C05411=1051.547,373.065,-118.694,173.770,40.070,157.709
C05412=1051.539,372.818,-118.654,173.765,40.065,157.708
C05413=1051.531,372.572,-118.614,173.759,40.059,157.706
C05414=1051.524,372.325,-118.575,173.753,40.054,157.704
C05415=1051.517,372.078,-118.535,173.748,40.048,157.703
C05416=1051.509,371.831,-118.495,173.742,40.043,157.701
C05417=1051.502,371.585,-118.455,173.737,40.037,157.700
C05418=1051.493,371.338,-118.416,173.731,40.032,157.698
C05419=1051.486,371.091,-118.376,173.726,40.027,157.697
C05420=1051.478,370.845,-118.336,173.720,40.021,157.695
C05421=1051.470,370.598,-118.298,173.714,40.015,157.694
C05422=1051.463,370.351,-118.258,173.709,40.010,157.692
C05423=1051.454,370.105,-118.219,173.703,40.005,157.691
C05424=1051.447,369.858,-118.180,173.698,40.000,157.689
C05425=1051.440,369.611,-118.140,173.692,39.994,157.688
C05426=1051.432,369.365,-118.101,173.687,39.989,157.686
C05427=1051.424,369.117,-118.062,173.681,39.984,157.685
C05428=1051.417,368.870,-118.022,173.676,39.978,157.683
C05429=1051.409,368.624,-117.984,173.670,39.974,157.682
C05430=1051.401,368.377,-117.944,173.665,39.968,157.680
C05431=1051.394,368.131,-117.905,173.659,39.963,157.679
C05432=1051.386,367.884,-117.865,173.654,39.958,157.677
C05433=1051.379,367.637,-117.827,173.648,39.952,157.676
C05434=1051.371,367.390,-117.787,173.643,39.947,157.674
C05435=1051.364,367.143,-117.748,173.637,39.942,157.673
C05436=1051.356,366.897,-117.709,173.632,39.937,157.672
C05437=1051.349,366.650,-117.670,173.626,39.931,157.670
C05438=1051.341,366.403,-117.632,173.621,39.926,157.669
C05439=1051.333,366.157,-117.592,173.615,39.921,157.667
C05440=1051.325,365.909,-117.554,173.610,39.916,157.666
C05441=1051.319,365.663,-117.515,173.604,39.911,157.664
C05442=1051.311,365.415,-117.475,173.599,39.906,157.663
C05443=1051.303,365.169,-117.437,173.594,39.900,157.661
C05444=1051.296,364.922,-117.398,173.589,39.895,157.660
C05445=1051.288,364.675,-117.359,173.584,39.890,157.659
C05446=1051.281,364.428,-117.320,173.578,39.885,157.657
C05447=1051.274,364.182,-117.282,173.573,39.880,157.656
C05448=1051.267,363.934,-117.243,173.567,39.875,157.654
C05449=1051.259,363.688,-117.205,173.562,39.870,157.653
C05450=1051.252,363.441,-117.166,173.557,39.865,157.651
C05451=1051.244,363.194,-117.127,173.552,39.860,157.650
C05452=1051.237,362.947,-117.088,173.547,39.855,157.649
C05453=1051.229,362.700,-117.050,173.541,39.850,157.647
C05454=1051.221,362.453,-117.011,173.536,39.845,157.646
C05455=1051.215,362.206,-116.973,173.530,39.840,157.644
C05456=1051.207,361.960,-116.934,173.526,39.835,157.643
C05457=1051.199,361.713,-116.896,173.521,39.830,157.642
C05458=1051.192,361.466,-116.857,173.515,39.825,157.640
C05459=1051.184,361.173,-116.812,173.509,39.819,157.639
C05460=1051.174,360.880,-116.766,173.503,39.813,157.637
C05461=1051.165,360.587,-116.721,173.496,39.808,157.636
C05462=1051.156,360.295,-116.676,173.491,39.802,157.634
C05463=1051.149,360.048,-116.638,173.485,39.797,157.633
C05464=1051.142,359.801,-116.599,173.480,39.792,157.631
C05465=1051.134,359.554,-116.561,173.476,39.787,157.630
C05466=1051.127,359.307,-116.523,173.470,39.782,157.629
C05467=1051.119,359.060,-116.485,173.465,39.777,157.627
C05468=1051.112,358.813,-116.447,173.460,39.773,157.626
C05469=1051.105,358.566,-116.409,173.455,39.768,157.625
C05470=1051.098,358.320,-116.370,173.450,39.763,157.623
C05471=1051.090,358.072,-116.333,173.445,39.758,157.622
C05472=1051.083,357.825,-116.295,173.440,39.753,157.621
C05473=1051.075,357.578,-116.257,173.435,39.748,157.619
C05474=1051.069,357.331,-116.219,173.430,39.744,157.618
C05475=1051.061,357.084,-116.180,173.424,39.739,157.617
C05476=1051.054,356.837,-116.143,173.420,39.734,157.615
C05477=1051.047,356.590,-116.105,173.415,39.729,157.614
C05478=1051.039,356.344,-116.067,173.410,39.725,157.613
C05479=1051.032,356.096,-116.030,173.405,39.720,157.612
C05480=1051.024,355.849,-115.992,173.400,39.715,157.610
C05481=1051.017,355.601,-115.954,173.395,39.710,157.609
C05482=1051.009,355.355,-115.916,173.391,39.706,157.608
C05483=1051.002,355.108,-115.878,173.385,39.701,157.606
C05484=1050.995,354.861,-115.841,173.380,39.696,157.605
C05485=1050.988,354.614,-115.803,173.376,39.692,157.604
C05486=1050.980,354.366,-115.766,173.370,39.687,157.603
C05487=1050.973,354.119,-115.728,173.365,39.682,157.601
C05488=1050.965,353.873,-115.690,173.361,39.678,157.600
C05489=1050.958,353.626,-115.652,173.356,39.673,157.599
C05490=1050.951,353.378,-115.615,173.350,39.668,157.597
C05491=1050.944,353.131,-115.577,173.346,39.664,157.596
C05492=1050.937,352.884,-115.540,173.341,39.659,157.595
C05493=1050.930,352.638,-115.503,173.337,39.655,157.594
C05494=1050.923,352.391,-115.465,173.331,39.650,157.592
C05495=1050.915,352.143,-115.428,173.326,39.646,157.591
C05496=1050.908,351.896,-115.390,173.322,39.641,157.590
C05497=1050.900,351.649,-115.354,173.317,39.637,157.589
C05498=1050.893,351.402,-115.316,173.312,39.632,157.587
C05499=1050.886,351.155,-115.279,173.307,39.627,157.586
C05500=1050.879,350.908,-115.241,173.303,39.622,157.585
C05501=1050.872,350.661,-115.204,173.298,39.618,157.584
C05502=1050.865,350.414,-115.167,173.293,39.614,157.583
C05503=1050.858,350.166,-115.130,173.288,39.609,157.581
C05504=1050.850,349.919,-115.093,173.283,39.605,157.580
C05505=1050.843,349.672,-115.055,173.279,39.600,157.579
C05506=1050.836,349.424,-115.019,173.274,39.596,157.578
C05507=1050.828,349.177,-114.981,173.270,39.591,157.576
C05508=1050.821,348.931,-114.945,173.264,39.587,157.575
C05509=1050.814,348.683,-114.908,173.260,39.582,157.574
C05510=1050.807,348.436,-114.870,173.255,39.578,157.573
C05511=1050.799,348.189,-114.834,173.251,39.574,157.572
C05512=1050.792,347.942,-114.796,173.246,39.569,157.570
C05513=1050.786,347.695,-114.760,173.242,39.565,157.569
C05514=1050.778,347.448,-114.722,173.236,39.560,157.568
C05515=1050.770,347.160,-114.680,173.231,39.555,157.567
C05516=1050.761,346.873,-114.637,173.226,39.550,157.565
C05517=1050.753,346.585,-114.594,173.220,39.545,157.564
C05518=1050.745,346.298,-114.552,173.215,39.540,157.563
C05519=1050.738,346.051,-114.514,173.210,39.535,157.561
C05520=1050.731,345.804,-114.478,173.206,39.531,157.560
C05521=1050.724,345.556,-114.441,173.202,39.527,157.559
C05522=1050.716,345.309,-114.405,173.196,39.522,157.558
C05523=1050.709,345.062,-114.368,173.192,39.518,157.557
C05524=1050.703,344.814,-114.331,173.187,39.514,157.556
C05525=1050.695,344.567,-114.295,173.183,39.509,157.554
C05526=1050.688,344.321,-114.258,173.178,39.506,157.553
C05527=1050.681,344.073,-114.221,173.174,39.501,157.552
C05528=1050.674,343.825,-114.185,173.169,39.497,157.551
C05529=1050.667,343.578,-114.148,173.165,39.493,157.550
C05530=1050.660,343.331,-114.112,173.161,39.488,157.549
C05531=1050.653,343.084,-114.075,173.155,39.484,157.548
C05532=1050.645,342.837,-114.039,173.151,39.479,157.546
C05533=1050.639,342.590,-114.002,173.146,39.475,157.545
C05534=1050.631,342.343,-113.966,173.142,39.471,157.544
C05535=1050.624,342.095,-113.929,173.138,39.467,157.543
C05536=1050.617,341.848,-113.893,173.133,39.463,157.542
C05537=1050.610,341.601,-113.857,173.129,39.458,157.541
C05538=1050.603,341.354,-113.821,173.124,39.455,157.540
C05539=1050.596,341.106,-113.785,173.120,39.450,157.539
C05540=1050.589,340.859,-113.748,173.116,39.446,157.537
C05541=1050.582,340.611,-113.713,173.111,39.442,157.536
C05542=1050.575,340.364,-113.677,173.106,39.438,157.535
C05543=1050.568,340.116,-113.640,173.102,39.433,157.534
C05544=1050.561,339.870,-113.604,173.097,39.430,157.533
C05545=1050.553,339.622,-113.568,173.093,39.425,157.532
C05546=1050.547,339.375,-113.531,173.089,39.421,157.531
C05547=1050.539,339.127,-113.496,173.084,39.417,157.530
C05548=1050.532,338.880,-113.460,173.080,39.413,157.529
C05549=1050.525,338.633,-113.423,173.076,39.409,157.528
C05550=1050.518,338.386,-113.387,173.071,39.404,157.526
C05551=1050.511,338.138,-113.352,173.067,39.401,157.525
C05552=1050.505,337.891,-113.316,173.063,39.396,157.524
C05553=1050.498,337.644,-113.280,173.058,39.392,157.523
C05554=1050.490,337.396,-113.244,173.054,39.388,157.522
C05555=1050.484,337.149,-113.208,173.050,39.384,157.521
C05556=1050.477,336.902,-113.172,173.046,39.380,157.520
C05557=1050.469,336.654,-113.136,173.041,39.376,157.519
C05558=1050.462,336.407,-113.101,173.037,39.372,157.518
C05559=1050.456,336.160,-113.065,173.033,39.368,157.517
C05560=1050.449,335.912,-113.029,173.028,39.364,157.516
C05561=1050.442,335.665,-112.993,173.024,39.360,157.514
C05562=1050.434,335.417,-112.957,173.020,39.356,157.513
C05563=1050.427,335.170,-112.922,173.016,39.352,157.512
C05564=1050.421,334.923,-112.887,173.011,39.348,157.511
C05565=1050.413,334.675,-112.851,173.007,39.344,157.510
C05566=1050.406,334.428,-112.816,173.003,39.340,157.509
C05567=1050.399,334.181,-112.780,172.999,39.336,157.508
C05568=1050.392,333.933,-112.744,172.994,39.332,157.507
C05569=1050.386,333.685,-112.709,172.990,39.328,157.506
C05570=1050.379,333.439,-112.673,172.986,39.324,157.505
C05571=1050.370,333.147,-112.632,172.980,39.319,157.504
C05572=1050.362,332.856,-112.590,172.975,39.315,157.503
C05573=1050.354,332.564,-112.548,172.971,39.310,157.501
C05574=1050.346,332.273,-112.506,172.966,39.306,157.500
C05575=1050.339,332.025,-112.471,172.962,39.302,157.499
C05576=1050.332,331.778,-112.435,172.957,39.297,157.498
C05577=1050.325,331.531,-112.400,172.953,39.293,157.497
C05578=1050.318,331.283,-112.365,172.949,39.290,157.496
C05579=1050.311,331.036,-112.329,172.945,39.286,157.495
C05580=1050.304,330.788,-112.294,172.941,39.282,157.494
C05581=1050.297,330.541,-112.259,172.936,39.278,157.493
C05582=1050.290,330.294,-112.224,172.932,39.274,157.492
C05583=1050.284,330.046,-112.188,172.928,39.270,157.491
C05584=1050.277,329.799,-112.153,172.924,39.266,157.490
C05585=1050.270,329.552,-112.118,172.920,39.262,157.489
C05586=1050.263,329.303,-112.083,172.916,39.258,157.488
C05587=1050.255,329.056,-112.048,172.911,39.255,157.487
C05588=1050.249,328.809,-112.013,172.907,39.251,157.486
C05589=1050.242,328.561,-111.979,172.903,39.247,157.485
C05590=1050.235,328.314,-111.944,172.900,39.244,157.484
C05591=1050.228,328.067,-111.909,172.896,39.240,157.483
C05592=1050.220,327.819,-111.874,172.892,39.236,157.482
C05593=1050.213,327.572,-111.839,172.887,39.232,157.481
C05594=1050.206,327.324,-111.804,172.883,39.229,157.480
C05595=1050.199,327.077,-111.770,172.879,39.225,157.479
C05596=1050.192,326.829,-111.735,172.875,39.221,157.478
C05597=1050.185,326.582,-111.700,172.871,39.217,157.477
C05598=1050.178,326.334,-111.666,172.867,39.213,157.476
C05599=1050.171,326.087,-111.631,172.863,39.210,157.475
C05600=1050.165,325.839,-111.595,172.859,39.206,157.474
C05601=1050.157,325.592,-111.562,172.854,39.202,157.473
C05602=1050.150,325.344,-111.526,172.850,39.199,157.472
C05603=1050.143,325.097,-111.492,172.847,39.195,157.471
C05604=1050.136,324.849,-111.457,172.843,39.191,157.470
C05605=1050.129,324.601,-111.422,172.839,39.188,157.469
C05606=1050.122,324.354,-111.388,172.835,39.184,157.468
C05607=1050.115,324.106,-111.353,172.831,39.180,157.467
C05608=1050.108,323.859,-111.319,172.827,39.177,157.467
C05609=1050.101,323.611,-111.284,172.823,39.173,157.466
C05610=1050.095,323.364,-111.249,172.819,39.169,157.465
C05611=1050.088,323.117,-111.216,172.815,39.166,157.464
C05612=1050.081,322.869,-111.180,172.811,39.162,157.463
C05613=1050.074,322.622,-111.147,172.808,39.158,157.462
C05614=1050.068,322.374,-111.112,172.804,39.154,157.461
C05615=1050.061,322.126,-111.077,172.800,39.151,157.460
C05616=1050.054,321.879,-111.043,172.795,39.147,157.459
C05617=1050.047,321.631,-111.008,172.791,39.144,157.458
C05618=1050.040,321.384,-110.974,172.787,39.140,157.457
C05619=1050.033,321.136,-110.940,172.783,39.136,157.456
C05620=1050.026,320.889,-110.905,172.779,39.132,157.455
C05621=1050.020,320.641,-110.871,172.775,39.129,157.454
C05622=1050.013,320.394,-110.837,172.772,39.125,157.453
C05623=1050.006,320.146,-110.802,172.768,39.121,157.452
C05624=1049.999,319.898,-110.768,172.764,39.118,157.451
C05625=1049.992,319.651,-110.734,172.760,39.114,157.450
C05626=1049.986,319.403,-110.700,172.756,39.110,157.449
C05627=1049.978,319.107,-110.659,172.752,39.106,157.448
C05628=1049.970,318.811,-110.618,172.747,39.102,157.447
C05629=1049.962,318.514,-110.576,172.743,39.098,157.446
C05630=1049.954,318.217,-110.536,172.738,39.093,157.445
C05631=1049.946,317.970,-110.501,172.734,39.090,157.444
C05632=1049.940,317.723,-110.467,172.730,39.086,157.443
C05633=1049.933,317.475,-110.434,172.727,39.083,157.442
C05634=1049.927,317.227,-110.399,172.723,39.079,157.441
C05635=1049.920,316.979,-110.365,172.720,39.075,157.440
C05636=1049.914,316.732,-110.331,172.716,39.072,157.439
C05637=1049.906,316.485,-110.297,172.712,39.068,157.439
C05638=1049.900,316.237,-110.263,172.708,39.064,157.438
C05639=1049.893,315.990,-110.230,172.704,39.061,157.437
C05640=1049.887,315.742,-110.195,172.700,39.057,157.436
C05641=1049.880,315.494,-110.161,172.697,39.054,157.435
C05642=1049.874,315.247,-110.127,172.693,39.050,157.434
C05643=1049.867,314.999,-110.093,172.689,39.047,157.433
C05644=1049.861,314.752,-110.059,172.685,39.043,157.432
C05645=1049.854,314.504,-110.026,172.681,39.039,157.431
C05646=1049.847,314.256,-109.991,172.678,39.035,157.430
C05647=1049.841,314.009,-109.958,172.675,39.032,157.429
C05648=1049.834,313.761,-109.923,172.671,39.029,157.429
C05649=1049.827,313.514,-109.890,172.667,39.025,157.428
C05650=1049.821,313.266,-109.855,172.663,39.022,157.427
C05651=1049.815,313.019,-109.823,172.659,39.018,157.426
C05652=1049.808,312.771,-109.789,172.655,39.014,157.425
C05653=1049.800,312.523,-109.755,172.652,39.011,157.424
C05654=1049.794,312.276,-109.722,172.648,39.008,157.423
C05655=1049.787,312.028,-109.688,172.645,39.004,157.422
C05656=1049.780,311.780,-109.655,172.641,39.001,157.421
C05657=1049.773,311.533,-109.622,172.637,38.997,157.420
C05658=1049.766,311.285,-109.588,172.634,38.994,157.420
C05659=1049.759,311.037,-109.555,172.630,38.991,157.419
C05660=1049.753,310.790,-109.521,172.626,38.987,157.418
C05661=1049.745,310.542,-109.488,172.622,38.984,157.417
C05662=1049.739,310.294,-109.455,172.618,38.981,157.416
C05663=1049.732,310.047,-109.421,172.616,38.977,157.415
C05664=1049.726,309.799,-109.388,172.612,38.974,157.415
C05665=1049.718,309.552,-109.355,172.608,38.971,157.414
C05666=1049.711,309.303,-109.322,172.604,38.967,157.413
C05667=1049.704,309.057,-109.289,172.601,38.964,157.412
C05668=1049.697,308.808,-109.255,172.597,38.961,157.411
C05669=1049.691,308.561,-109.222,172.593,38.957,157.410
C05670=1049.684,308.313,-109.189,172.590,38.953,157.409
C05671=1049.678,308.065,-109.156,172.586,38.950,157.408
C05672=1049.670,307.818,-109.122,172.583,38.947,157.408
C05673=1049.664,307.570,-109.090,172.579,38.943,157.407
C05674=1049.656,307.322,-109.057,172.575,38.940,157.406
C05675=1049.650,307.075,-109.024,172.571,38.937,157.405
C05676=1049.644,306.828,-108.991,172.569,38.933,157.404
C05677=1049.637,306.579,-108.958,172.565,38.930,157.403
C05678=1049.630,306.332,-108.924,172.561,38.927,157.403
C05679=1049.623,306.084,-108.891,172.557,38.923,157.402
C05680=1049.617,305.836,-108.858,172.553,38.920,157.401
C05681=1049.610,305.589,-108.825,172.551,38.917,157.400
C05682=1049.603,305.341,-108.792,172.547,38.913,157.399
C05683=1049.595,305.049,-108.753,172.543,38.909,157.398
C05684=1049.587,304.757,-108.714,172.538,38.905,157.397
C05685=1049.580,304.466,-108.676,172.534,38.901,157.396
C05686=1049.571,304.174,-108.637,172.530,38.898,157.395
C05687=1049.564,303.925,-108.604,172.527,38.894,157.394
C05688=1049.558,303.678,-108.571,172.523,38.891,157.394
C05689=1049.552,303.430,-108.538,172.520,38.887,157.393
C05690=1049.545,303.182,-108.505,172.516,38.884,157.392
C05691=1049.539,302.934,-108.473,172.513,38.881,157.391
C05692=1049.532,302.687,-108.440,172.509,38.877,157.390
C05693=1049.525,302.439,-108.407,172.506,38.875,157.389
C05694=1049.518,302.191,-108.375,172.502,38.871,157.389
C05695=1049.512,301.943,-108.342,172.499,38.868,157.388
C05696=1049.506,301.696,-108.309,172.495,38.865,157.387
C05697=1049.499,301.448,-108.276,172.492,38.861,157.386
C05698=1049.493,301.200,-108.243,172.488,38.858,157.385
C05699=1049.486,300.953,-108.211,172.485,38.854,157.384
C05700=1049.479,300.705,-108.178,172.482,38.851,157.384
C05701=1049.472,300.457,-108.145,172.478,38.848,157.383
C05702=1049.466,300.209,-108.113,172.474,38.844,157.382
C05703=1049.460,299.962,-108.080,172.472,38.841,157.381
C05704=1049.453,299.714,-108.048,172.468,38.838,157.380
C05705=1049.446,299.467,-108.015,172.464,38.835,157.380
C05706=1049.440,299.218,-107.982,172.461,38.831,157.379
C05707=1049.433,298.971,-107.949,172.458,38.828,157.378
C05708=1049.427,298.723,-107.916,172.454,38.825,157.377
C05709=1049.420,298.475,-107.885,172.451,38.821,157.376
C05710=1049.414,298.228,-107.852,172.447,38.818,157.375
C05711=1049.408,297.980,-107.819,172.444,38.815,157.375
C05712=1049.401,297.733,-107.787,172.441,38.812,157.374
C05713=1049.394,297.484,-107.754,172.437,38.808,157.373
C05714=1049.388,297.236,-107.722,172.433,38.805,157.372
C05715=1049.381,296.989,-107.689,172.431,38.802,157.371
C05716=1049.375,296.741,-107.657,172.427,38.798,157.370
C05717=1049.369,296.493,-107.625,172.424,38.795,157.370
C05718=1049.362,296.246,-107.592,172.421,38.792,157.369
C05719=1049.356,295.998,-107.560,172.417,38.789,157.368
C05720=1049.350,295.750,-107.528,172.414,38.785,157.367
C05721=1049.342,295.502,-107.495,172.410,38.782,157.366
C05722=1049.336,295.254,-107.462,172.407,38.779,157.366
C05723=1049.329,295.006,-107.431,172.404,38.776,157.365
C05724=1049.323,294.759,-107.398,172.400,38.772,157.364
C05725=1049.316,294.511,-107.367,172.398,38.770,157.363
C05726=1049.309,294.264,-107.335,172.394,38.766,157.363
C05727=1049.303,294.015,-107.303,172.390,38.763,157.362
C05728=1049.296,293.768,-107.270,172.388,38.760,157.361
C05729=1049.290,293.520,-107.238,172.384,38.757,157.360
C05730=1049.283,293.271,-107.207,172.381,38.753,157.359
C05731=1049.276,293.024,-107.174,172.377,38.750,157.359
C05732=1049.270,292.776,-107.142,172.374,38.747,157.358
C05733=1049.263,292.529,-107.110,172.371,38.744,157.357
C05734=1049.256,292.281,-107.079,172.367,38.741,157.356
C05735=1049.250,292.032,-107.047,172.365,38.737,157.355
C05736=1049.243,291.785,-107.015,172.361,38.735,157.355
C05737=1049.237,291.537,-106.983,172.357,38.731,157.354
C05738=1049.230,291.289,-106.951,172.355,38.729,157.353
C05739=1049.223,291.013,-106.915,172.351,38.725,157.352
C05740=1049.216,290.737,-106.880,172.347,38.721,157.351
C05741=1049.208,290.462,-106.845,172.343,38.718,157.351
C05742=1049.201,290.186,-106.810,172.340,38.714,157.350
C05743=1049.194,289.938,-106.778,172.337,38.711,157.349
C05744=1049.188,289.689,-106.746,172.333,38.708,157.348
C05745=1049.181,289.442,-106.714,172.330,38.705,157.347
C05746=1049.174,289.194,-106.682,172.327,38.702,157.347
C05747=1049.168,288.946,-106.651,172.324,38.699,157.346
C05748=1049.162,288.698,-106.619,172.320,38.696,157.345
C05749=1049.155,288.450,-106.588,172.318,38.692,157.344
C05750=1049.148,288.202,-106.556,172.314,38.690,157.344
C05751=1049.141,287.955,-106.524,172.311,38.686,157.343
C05752=1049.135,287.707,-106.492,172.308,38.683,157.342
C05753=1049.129,287.459,-106.461,172.305,38.680,157.341
C05754=1049.122,287.211,-106.429,172.301,38.677,157.341
C05755=1049.115,286.963,-106.398,172.299,38.674,157.340
C05756=1049.108,286.715,-106.366,172.295,38.671,157.339
C05757=1049.102,286.467,-106.335,172.292,38.667,157.338
C05758=1049.095,286.219,-106.303,172.289,38.665,157.338
C05759=1049.085,285.816,-106.253,172.284,38.660,157.336
C05760=1049.074,285.412,-106.201,172.279,38.654,157.335
C05761=1049.063,285.009,-106.150,172.274,38.650,157.334
C05762=1049.052,284.605,-106.100,172.268,38.645,157.333
C05763=1049.045,284.358,-106.068,172.265,38.641,157.332
C05764=1049.039,284.109,-106.036,172.262,38.639,157.331
C05765=1049.033,283.861,-106.005,172.259,38.636,157.331
C05766=1049.026,283.613,-105.974,172.256,38.632,157.330
C05767=1049.020,283.365,-105.943,172.252,38.630,157.329
C05768=1049.013,283.117,-105.911,172.249,38.626,157.328
C05769=1049.007,282.870,-105.880,172.247,38.623,157.327
C05770=1049.000,282.622,-105.849,172.243,38.621,157.327
C05771=1048.994,282.373,-105.818,172.241,38.617,157.326
C05772=1048.987,282.126,-105.787,172.237,38.614,157.325
C05773=1048.980,281.878,-105.755,172.234,38.611,157.324
C05774=1048.974,281.630,-105.724,172.231,38.608,157.324
C05775=1048.968,281.382,-105.694,172.228,38.605,157.323
C05776=1048.961,281.134,-105.662,172.224,38.602,157.322
C05777=1048.954,280.886,-105.631,172.222,38.599,157.322
C05778=1048.948,280.638,-105.600,172.219,38.595,157.321
C05779=1048.942,280.390,-105.569,172.215,38.593,157.320
C05780=1048.935,280.142,-105.537,172.213,38.590,157.319
C05781=1048.928,279.894,-105.507,172.209,38.586,157.319
C05782=1048.922,279.646,-105.475,172.206,38.584,157.318
C05783=1048.916,279.398,-105.445,172.204,38.580,157.317
C05784=1048.909,279.150,-105.414,172.200,38.577,157.316
C05785=1048.902,278.902,-105.383,172.198,38.574,157.316
C05786=1048.895,278.654,-105.352,172.194,38.572,157.315
C05787=1048.889,278.406,-105.322,172.191,38.568,157.314
C05788=1048.883,278.158,-105.290,172.189,38.565,157.313
C05789=1048.876,277.910,-105.259,172.185,38.563,157.313
C05790=1048.869,277.662,-105.229,172.182,38.560,157.312
C05791=1048.860,277.305,-105.185,172.177,38.555,157.311
C05792=1048.851,276.949,-105.141,172.174,38.551,157.310
C05793=1048.842,276.592,-105.096,172.170,38.547,157.309
C05794=1048.832,276.235,-105.052,172.165,38.542,157.308
C05795=1048.825,275.987,-105.021,172.162,38.539,157.307
C05796=1048.819,275.739,-104.990,172.159,38.536,157.306
C05797=1048.813,275.491,-104.960,172.156,38.533,157.306
C05798=1048.806,275.243,-104.928,172.153,38.530,157.305
C05799=1048.799,274.995,-104.899,172.150,38.527,157.304
C05800=1048.793,274.747,-104.868,172.147,38.524,157.304
C05801=1048.786,274.499,-104.836,172.144,38.521,157.303
C05802=1048.780,274.251,-104.807,172.141,38.518,157.302
C05803=1048.773,274.003,-104.776,172.138,38.515,157.301
C05804=1048.767,273.754,-104.745,172.136,38.512,157.301
C05805=1048.760,273.507,-104.715,172.132,38.509,157.300
C05806=1048.753,273.259,-104.684,172.129,38.506,157.299
C05807=1048.747,273.010,-104.653,172.127,38.503,157.299
C05808=1048.741,272.763,-104.624,172.123,38.500,157.298
C05809=1048.734,272.514,-104.593,172.120,38.497,157.297
C05810=1048.728,272.267,-104.563,172.118,38.494,157.296
C05811=1048.721,272.019,-104.532,172.114,38.491,157.296
C05812=1048.714,271.770,-104.501,172.112,38.488,157.295
C05813=1048.708,271.523,-104.471,172.109,38.485,157.294
C05814=1048.701,271.274,-104.440,172.106,38.483,157.294
C05815=1048.695,271.026,-104.410,172.103,38.480,157.293
C05816=1048.688,270.778,-104.380,172.100,38.476,157.292
C05817=1048.682,270.530,-104.349,172.098,38.473,157.291
C05818=1048.675,270.282,-104.320,172.094,38.471,157.291
C05819=1048.669,270.034,-104.289,172.091,38.468,157.290
C05820=1048.662,269.786,-104.259,172.089,38.465,157.289
C05821=1048.656,269.538,-104.228,172.085,38.462,157.289
C05822=1048.649,269.290,-104.198,172.082,38.459,157.288
C05823=1048.643,269.042,-104.168,172.080,38.456,157.287
C05824=1048.636,268.794,-104.138,172.077,38.453,157.287
C05825=1048.630,268.546,-104.107,172.074,38.450,157.286
C05826=1048.623,268.297,-104.077,172.071,38.447,157.285
C05827=1048.617,268.050,-104.047,172.069,38.444,157.284
C05828=1048.610,267.801,-104.018,172.066,38.441,157.284
C05829=1048.604,267.553,-103.988,172.062,38.438,157.283
C05830=1048.597,267.305,-103.957,172.060,38.435,157.282
C05831=1048.591,267.057,-103.927,172.057,38.432,157.282
C05832=1048.584,266.809,-103.897,172.055,38.429,157.281
C05833=1048.578,266.561,-103.868,172.051,38.426,157.280
C05834=1048.571,266.312,-103.837,172.048,38.424,157.280
C05835=1048.564,266.065,-103.808,172.046,38.421,157.279
C05836=1048.558,265.816,-103.777,172.043,38.418,157.278
C05837=1048.551,265.569,-103.747,172.040,38.415,157.278
C05838=1048.545,265.320,-103.717,172.037,38.412,157.277
C05839=1048.539,265.072,-103.687,172.034,38.409,157.276
C05840=1048.532,264.824,-103.657,172.032,38.406,157.275
C05841=1048.526,264.576,-103.628,172.029,38.403,157.275
C05842=1048.519,264.327,-103.598,172.026,38.400,157.274
C05843=1048.512,264.080,-103.568,172.023,38.397,157.273
C05844=1048.506,263.831,-103.538,172.020,38.394,157.273
C05845=1048.500,263.583,-103.508,172.018,38.391,157.272
C05846=1048.493,263.336,-103.478,172.015,38.388,157.271
C05847=1048.486,263.075,-103.447,172.012,38.385,157.271
C05848=1048.480,262.814,-103.416,172.009,38.382,157.270
C05849=1048.473,262.555,-103.385,172.006,38.379,157.269
C05850=1048.466,262.294,-103.354,172.003,38.376,157.268
C05851=1048.459,262.046,-103.324,172.000,38.374,157.268
C05852=1048.453,261.798,-103.295,171.998,38.371,157.267
C05853=1048.446,261.550,-103.264,171.995,38.368,157.266
C05854=1048.439,261.302,-103.235,171.992,38.365,157.266
C05855=1048.433,261.054,-103.206,171.989,38.362,157.265
C05856=1048.426,260.805,-103.176,171.986,38.359,157.264
C05857=1048.419,260.558,-103.146,171.984,38.356,157.264
C05858=1048.413,260.309,-103.117,171.981,38.353,157.263
C05859=1048.406,260.061,-103.088,171.979,38.351,157.262
C05860=1048.399,259.813,-103.058,171.975,38.348,157.262
C05861=1048.393,259.564,-103.029,171.973,38.345,157.261
C05862=1048.386,259.317,-103.000,171.970,38.342,157.260
C05863=1048.379,259.068,-102.970,171.967,38.339,157.260
C05864=1048.373,258.820,-102.941,171.965,38.336,157.259
C05865=1048.366,258.571,-102.912,171.962,38.333,157.258
C05866=1048.359,258.324,-102.882,171.959,38.330,157.258
C05867=1048.353,258.076,-102.853,171.956,38.327,157.257
C05868=1048.346,257.827,-102.824,171.954,38.325,157.256
C05869=1048.339,257.580,-102.794,171.951,38.322,157.256
C05870=1048.333,257.331,-102.765,171.949,38.319,157.255
C05871=1048.326,257.083,-102.735,171.946,38.317,157.254
C05872=1048.320,256.834,-102.706,171.943,38.314,157.254
C05873=1048.314,256.587,-102.677,171.940,38.311,157.253
C05874=1048.307,256.338,-102.647,171.937,38.308,157.252
C05875=1048.300,256.090,-102.618,171.935,38.305,157.252
C05876=1048.294,255.842,-102.589,171.932,38.302,157.251
C05877=1048.287,255.593,-102.560,171.930,38.299,157.250
C05878=1048.281,255.345,-102.530,171.927,38.296,157.250
C05879=1048.275,255.097,-102.501,171.925,38.293,157.249
C05880=1048.268,254.850,-102.472,171.922,38.290,157.248
C05881=1048.261,254.601,-102.443,171.919,38.288,157.248
C05882=1048.254,254.353,-102.414,171.916,38.285,157.247
C05883=1048.248,254.104,-102.385,171.913,38.282,157.246
C05884=1048.242,253.856,-102.356,171.911,38.279,157.246
C05885=1048.235,253.607,-102.327,171.908,38.276,157.245
C05886=1048.229,253.359,-102.298,171.906,38.273,157.244
C05887=1048.222,253.112,-102.268,171.903,38.270,157.244
C05888=1048.216,252.864,-102.239,171.900,38.267,157.243
C05889=1048.209,252.615,-102.209,171.898,38.264,157.242
C05890=1048.203,252.367,-102.180,171.895,38.262,157.242
C05891=1048.196,252.119,-102.152,171.893,38.259,157.241
C05892=1048.190,251.871,-102.123,171.890,38.256,157.240
C05893=1048.183,251.623,-102.094,171.888,38.253,157.240
C05894=1048.177,251.374,-102.064,171.885,38.250,157.239
C05895=1048.170,251.126,-102.035,171.883,38.247,157.238
C05896=1048.164,250.878,-102.006,171.880,38.244,157.238
C05897=1048.158,250.629,-101.977,171.876,38.241,157.237
C05898=1048.152,250.381,-101.949,171.874,38.238,157.236
C05899=1048.146,250.133,-101.920,171.871,38.235,157.236
C05900=1048.138,249.884,-101.891,171.869,38.233,157.235
C05901=1048.132,249.636,-101.862,171.866,38.230,157.234
C05902=1048.126,249.388,-101.833,171.864,38.227,157.234
C05903=1048.119,249.126,-101.802,171.861,38.224,157.233
C05904=1048.113,248.864,-101.772,171.858,38.220,157.232
C05905=1048.106,248.603,-101.741,171.856,38.217,157.231
C05906=1048.098,248.341,-101.711,171.853,38.214,157.231
C05907=1048.092,248.092,-101.683,171.851,38.212,157.230
C05908=1048.086,247.844,-101.653,171.848,38.209,157.229
C05909=1048.080,247.596,-101.624,171.846,38.206,157.229
C05910=1048.074,247.348,-101.595,171.843,38.203,157.228
C05911=1048.067,247.100,-101.566,171.841,38.200,157.227
C05912=1048.062,246.851,-101.538,171.838,38.196,157.227
C05913=1048.055,246.603,-101.510,171.835,38.194,157.226
C05914=1048.048,246.355,-101.481,171.833,38.191,157.225
C05915=1048.042,246.107,-101.451,171.830,38.188,157.225
C05916=1048.036,245.858,-101.423,171.828,38.185,157.224
C05917=1048.030,245.610,-101.394,171.825,38.182,157.223
C05918=1048.022,245.362,-101.365,171.823,38.179,157.223
C05919=1048.016,245.113,-101.337,171.820,38.176,157.222
C05920=1048.010,244.865,-101.308,171.817,38.173,157.221
C05921=1048.003,244.617,-101.280,171.815,38.170,157.221
C05922=1047.997,244.368,-101.251,171.812,38.168,157.220
C05923=1047.990,244.120,-101.223,171.810,38.165,157.219
C05924=1047.984,243.872,-101.194,171.807,38.162,157.219
C05925=1047.978,243.623,-101.165,171.805,38.159,157.218
C05926=1047.971,243.376,-101.137,171.803,38.156,157.217
C05927=1047.965,243.127,-101.109,171.801,38.153,157.217
C05928=1047.958,242.879,-101.080,171.798,38.150,157.216
C05929=1047.952,242.630,-101.052,171.796,38.147,157.215
C05930=1047.946,242.382,-101.023,171.793,38.145,157.215
C05931=1047.939,242.134,-100.995,171.791,38.142,157.214
C05932=1047.933,241.886,-100.966,171.788,38.139,157.213
C05933=1047.926,241.637,-100.938,171.785,38.136,157.213
C05934=1047.920,241.389,-100.909,171.783,38.133,157.212
C05935=1047.913,241.141,-100.882,171.780,38.130,157.211
C05936=1047.907,240.892,-100.853,171.778,38.127,157.211
C05937=1047.900,240.644,-100.825,171.775,38.124,157.210
C05938=1047.894,240.396,-100.797,171.773,38.121,157.209
C05939=1047.887,240.147,-100.768,171.770,38.119,157.209
C05940=1047.881,239.899,-100.740,171.768,38.116,157.208
C05941=1047.874,239.651,-100.713,171.766,38.113,157.208
C05942=1047.868,239.402,-100.683,171.764,38.110,157.207
C05943=1047.861,239.154,-100.656,171.761,38.107,157.206
C05944=1047.855,238.905,-100.627,171.759,38.104,157.206
C05945=1047.848,238.657,-100.599,171.756,38.101,157.205
C05946=1047.842,238.409,-100.571,171.753,38.098,157.204
C05947=1047.836,238.160,-100.543,171.751,38.095,157.204
C05948=1047.829,237.912,-100.515,171.748,38.093,157.203
C05949=1047.822,237.664,-100.487,171.746,38.090,157.202
C05950=1047.815,237.415,-100.459,171.743,38.087,157.202
C05951=1047.809,237.167,-100.431,171.742,38.084,157.201
C05952=1047.803,236.918,-100.403,171.739,38.081,157.200
C05953=1047.796,236.670,-100.375,171.737,38.078,157.200
C05954=1047.790,236.422,-100.346,171.734,38.076,157.199
C05955=1047.783,236.173,-100.318,171.732,38.073,157.198
C05956=1047.777,235.926,-100.291,171.729,38.070,157.198
C05957=1047.770,235.677,-100.263,171.727,38.067,157.197
C05958=1047.764,235.428,-100.235,171.724,38.064,157.197
C05959=1047.757,235.161,-100.205,171.722,38.061,157.196
C05960=1047.749,234.893,-100.175,171.719,38.058,157.195
C05961=1047.743,234.626,-100.145,171.716,38.055,157.195
C05962=1047.736,234.358,-100.115,171.714,38.052,157.194
C05963=1047.730,234.109,-100.087,171.712,38.049,157.193
C05964=1047.723,233.862,-100.059,171.710,38.046,157.192
C05965=1047.717,233.614,-100.031,171.707,38.043,157.192
C05966=1047.711,233.365,-100.003,171.705,38.040,157.191
C05967=1047.704,233.117,-99.975,171.702,38.037,157.191
C05968=1047.697,232.868,-99.947,171.701,38.034,157.190
C05969=1047.691,232.620,-99.920,171.698,38.032,157.189
C05970=1047.685,232.371,-99.891,171.696,38.029,157.189
C05971=1047.679,232.123,-99.864,171.693,38.026,157.188
C05972=1047.672,231.875,-99.836,171.691,38.023,157.187
C05973=1047.665,231.626,-99.808,171.688,38.020,157.187
C05974=1047.658,231.378,-99.781,171.687,38.017,157.186
C05975=1047.652,231.129,-99.753,171.684,38.014,157.185
C05976=1047.645,230.881,-99.725,171.681,38.011,157.185
C05977=1047.640,230.632,-99.698,171.679,38.008,157.184
C05978=1047.633,230.384,-99.670,171.676,38.005,157.183
C05979=1047.627,230.135,-99.642,171.675,38.002,157.183
C05980=1047.620,229.887,-99.615,171.672,38.000,157.182
C05981=1047.613,229.638,-99.587,171.670,37.997,157.181
C05982=1047.607,229.391,-99.560,171.667,37.994,157.181
C05983=1047.601,229.142,-99.532,171.665,37.991,157.180
C05984=1047.594,228.894,-99.504,171.663,37.988,157.180
C05985=1047.588,228.645,-99.477,171.661,37.985,157.179
C05986=1047.581,228.397,-99.450,171.658,37.982,157.178
C05987=1047.575,228.149,-99.422,171.656,37.979,157.178
C05988=1047.568,227.900,-99.394,171.653,37.976,157.177
C05989=1047.562,227.651,-99.367,171.652,37.974,157.176
C05990=1047.555,227.403,-99.340,171.649,37.971,157.176
C05991=1047.549,227.155,-99.312,171.647,37.968,157.175
C05992=1047.542,226.907,-99.285,171.644,37.965,157.174
C05993=1047.535,226.658,-99.258,171.643,37.962,157.174
C05994=1047.528,226.409,-99.230,171.640,37.959,157.173
C05995=1047.522,226.161,-99.203,171.638,37.956,157.172
C05996=1047.516,225.913,-99.176,171.635,37.953,157.172
C05997=1047.509,225.664,-99.148,171.634,37.950,157.171
C05998=1047.503,225.416,-99.121,171.631,37.948,157.171
C05999=1047.497,225.167,-99.094,171.629,37.945,157.170
C06000=1047.490,224.919,-99.066,171.626,37.942,157.169
C06001=1047.484,224.670,-99.039,171.625,37.939,157.169
C06002=1047.476,224.422,-99.012,171.622,37.936,157.168
C06003=1047.470,224.174,-98.985,171.620,37.933,157.167
C06004=1047.464,223.925,-98.958,171.617,37.930,157.167
C06005=1047.457,223.676,-98.930,171.616,37.927,157.166
C06006=1047.452,223.428,-98.903,171.613,37.924,157.165
C06007=1047.445,223.180,-98.875,171.611,37.921,157.165
C06008=1047.438,222.931,-98.848,171.609,37.918,157.164
C06009=1047.432,222.683,-98.822,171.606,37.916,157.163
C06010=1047.425,222.435,-98.794,171.604,37.913,157.163
C06011=1047.419,222.186,-98.767,171.602,37.910,157.162
C06012=1047.412,221.938,-98.740,171.600,37.907,157.162
C06013=1047.406,221.689,-98.713,171.598,37.904,157.161
C06014=1047.399,221.440,-98.685,171.595,37.901,157.160
C06015=1047.392,221.165,-98.655,171.592,37.898,157.159
C06016=1047.385,220.890,-98.625,171.591,37.895,157.159
C06017=1047.378,220.615,-98.595,171.588,37.891,157.158
C06018=1047.371,220.340,-98.566,171.586,37.888,157.157
C06019=1047.365,220.092,-98.539,171.583,37.885,157.157
C06020=1047.358,219.844,-98.511,171.582,37.882,157.156
C06021=1047.351,219.595,-98.485,171.579,37.879,157.155
C06022=1047.345,219.346,-98.458,171.577,37.876,157.155
C06023=1047.338,219.098,-98.431,171.574,37.874,157.154
C06024=1047.331,218.849,-98.404,171.573,37.871,157.153
C06025=1047.326,218.601,-98.377,171.570,37.868,157.153
C06026=1047.318,218.353,-98.350,171.568,37.865,157.152
C06027=1047.312,218.104,-98.323,171.566,37.862,157.152
C06028=1047.305,217.856,-98.297,171.564,37.859,157.151
C06029=1047.299,217.607,-98.270,171.561,37.856,157.150
C06030=1047.293,217.359,-98.243,171.560,37.853,157.150
C06031=1047.286,217.110,-98.216,171.557,37.850,157.149
C06032=1047.279,216.861,-98.189,171.555,37.847,157.148
C06033=1047.273,216.613,-98.163,171.553,37.844,157.148
C06034=1047.266,216.365,-98.135,171.551,37.842,157.147
C06035=1047.260,216.116,-98.109,171.549,37.839,157.146
C06036=1047.253,215.867,-98.082,171.547,37.836,157.146
C06037=1047.248,215.619,-98.056,171.544,37.833,157.145
C06038=1047.240,215.371,-98.029,171.543,37.830,157.145
C06039=1047.234,215.122,-98.002,171.540,37.827,157.144
C06040=1047.227,214.874,-97.976,171.538,37.824,157.143
C06041=1047.221,214.625,-97.949,171.536,37.821,157.143
C06042=1047.214,214.377,-97.922,171.534,37.818,157.142
C06043=1047.208,214.128,-97.895,171.532,37.815,157.141
C06044=1047.202,213.880,-97.868,171.530,37.812,157.141
C06045=1047.195,213.631,-97.842,171.527,37.809,157.140
C06046=1047.189,213.383,-97.815,171.526,37.807,157.139
C06047=1047.182,213.134,-97.789,171.523,37.804,157.139
C06048=1047.176,212.886,-97.762,171.522,37.801,157.138
C06049=1047.169,212.637,-97.736,171.519,37.798,157.137
C06050=1047.163,212.389,-97.709,171.517,37.795,157.137
C06051=1047.156,212.140,-97.682,171.515,37.792,157.136
C06052=1047.150,211.891,-97.656,171.513,37.789,157.136
C06053=1047.143,211.643,-97.629,171.511,37.786,157.135
C06054=1047.137,211.394,-97.603,171.509,37.783,157.134
C06055=1047.130,211.146,-97.576,171.506,37.780,157.134
C06056=1047.124,210.898,-97.550,171.505,37.777,157.133
C06057=1047.117,210.648,-97.523,171.502,37.774,157.132
C06058=1047.111,210.400,-97.497,171.501,37.771,157.132
C06059=1047.105,210.151,-97.470,171.498,37.768,157.131
C06060=1047.098,209.903,-97.444,171.497,37.765,157.130
C06061=1047.092,209.655,-97.418,171.494,37.762,157.130
C06062=1047.085,209.406,-97.391,171.492,37.759,157.129
C06063=1047.079,209.158,-97.365,171.490,37.756,157.128
C06064=1047.072,208.909,-97.339,171.488,37.753,157.128
C06065=1047.066,208.661,-97.312,171.486,37.750,157.127
C06066=1047.059,208.412,-97.286,171.484,37.747,157.126
C06067=1047.052,208.164,-97.260,171.482,37.744,157.126
C06068=1047.046,207.915,-97.233,171.480,37.741,157.125
C06069=1047.040,207.667,-97.207,171.477,37.738,157.125
C06070=1047.033,207.418,-97.181,171.476,37.735,157.124
C06071=1047.026,207.148,-97.153,171.473,37.732,157.123
C06072=1047.019,206.879,-97.124,171.471,37.729,157.122
C06073=1047.011,206.610,-97.096,171.469,37.726,157.122
C06074=1047.004,206.339,-97.067,171.466,37.723,157.121
C06075=1046.978,205.288,-96.961,171.219,37.623,157.097
C06076=1046.972,205.039,-96.936,171.216,37.621,157.097
C06077=1046.966,204.791,-96.911,171.213,37.619,157.097
C06078=1046.960,204.542,-96.886,171.211,37.617,157.096
C06079=1046.954,204.293,-96.861,171.208,37.614,157.095
C06080=1046.948,204.044,-96.836,171.205,37.612,157.095
C06081=1046.942,203.796,-96.810,171.203,37.610,157.095
C06082=1046.936,203.547,-96.785,171.200,37.608,157.094
C06083=1046.930,203.298,-96.761,171.197,37.606,157.094
C06084=1046.924,203.050,-96.735,171.194,37.604,157.093
C06085=1046.918,202.801,-96.710,171.192,37.601,157.093
C06086=1046.911,202.553,-96.685,171.189,37.599,157.092
C06087=1046.906,202.304,-96.661,171.186,37.597,157.092
C06088=1046.900,202.056,-96.636,171.184,37.595,157.091
C06089=1046.893,201.807,-96.610,171.181,37.593,157.091
C06090=1046.887,201.558,-96.586,171.178,37.591,157.090
C06091=1046.881,201.309,-96.560,171.176,37.589,157.090
C06092=1046.876,201.060,-96.536,171.173,37.586,157.089
C06093=1046.869,200.812,-96.511,171.170,37.585,157.089
C06094=1046.863,200.563,-96.487,171.168,37.582,157.088
C06095=1046.856,200.314,-96.462,171.165,37.580,157.088
C06096=1046.850,200.065,-96.438,171.162,37.578,157.088
C06097=1046.845,199.817,-96.413,171.160,37.576,157.087
C06098=1046.838,199.568,-96.389,171.157,37.574,157.087
C06099=1046.832,199.319,-96.363,171.154,37.572,157.086
C06100=1046.825,199.070,-96.339,171.152,37.570,157.086
C06101=1046.819,198.822,-96.314,171.150,37.568,157.085
C06102=1046.814,198.573,-96.290,171.146,37.566,157.085
C06103=1046.807,198.325,-96.265,171.144,37.564,157.084
C06104=1046.801,198.076,-96.240,171.142,37.562,157.084
C06105=1046.794,197.827,-96.215,171.138,37.560,157.084
C06106=1046.789,197.579,-96.191,171.136,37.558,157.083
C06107=1046.782,197.330,-96.167,171.134,37.556,157.083
C06108=1046.776,197.081,-96.142,171.130,37.554,157.082
C06109=1046.770,196.832,-96.118,171.128,37.551,157.082
C06110=1046.764,196.584,-96.093,171.126,37.550,157.081
C06111=1046.758,196.335,-96.068,171.123,37.548,157.081
C06112=1046.752,196.086,-96.045,171.120,37.546,157.080
C06113=1046.745,195.838,-96.019,171.118,37.544,157.080
C06114=1046.739,195.589,-95.995,171.115,37.541,157.080
C06115=1046.733,195.340,-95.971,171.113,37.540,157.079
C06116=1046.727,195.092,-95.946,171.110,37.538,157.079
C06117=1046.721,194.843,-95.922,171.107,37.535,157.078
C06118=1046.715,194.594,-95.897,171.105,37.534,157.078
C06119=1046.709,194.345,-95.873,171.102,37.531,157.077
C06120=1046.702,194.096,-95.848,171.099,37.530,157.077
C06121=1046.696,193.848,-95.824,171.097,37.528,157.077
C06122=1046.691,193.599,-95.800,171.095,37.525,157.076
C06123=1046.684,193.350,-95.776,171.091,37.524,157.076
C06124=1046.678,193.102,-95.751,171.089,37.522,157.075
C06125=1046.672,192.853,-95.727,171.087,37.519,157.075
C06126=1046.666,192.604,-95.702,171.085,37.518,157.074
C06127=1046.660,192.355,-95.678,171.082,37.515,157.074
C06128=1046.654,192.106,-95.654,171.079,37.513,157.074
C06129=1046.648,191.858,-95.629,171.077,37.512,157.073
C06130=1046.642,191.609,-95.605,171.074,37.509,157.073
C06131=1046.636,191.360,-95.580,171.072,37.508,157.072
C06132=1046.630,191.111,-95.556,171.069,37.506,157.072
C06133=1046.624,190.863,-95.532,171.066,37.503,157.071
C06134=1046.618,190.614,-95.508,171.064,37.502,157.071
C06135=1046.612,190.365,-95.484,171.062,37.500,157.071
C06136=1046.605,190.081,-95.456,171.058,37.497,157.070
C06137=1046.598,189.796,-95.428,171.056,37.495,157.070
C06138=1046.591,189.512,-95.400,171.053,37.493,157.069
C06139=1046.584,189.228,-95.373,171.050,37.490,157.069
C06140=1046.578,188.979,-95.349,171.048,37.488,157.068
C06141=1046.572,188.730,-95.325,171.045,37.487,157.068
C06142=1046.566,188.481,-95.300,171.042,37.484,157.067
C06143=1046.560,188.233,-95.277,171.040,37.483,157.067
C06144=1046.554,187.983,-95.252,171.038,37.481,157.066
C06145=1046.548,187.735,-95.229,171.035,37.478,157.066
C06146=1046.542,187.486,-95.204,171.032,37.477,157.066
C06147=1046.536,187.238,-95.180,171.030,37.475,157.065
C06148=1046.531,186.988,-95.156,171.027,37.473,157.065
C06149=1046.524,186.740,-95.132,171.025,37.471,157.064
C06150=1046.519,186.491,-95.108,171.023,37.469,157.064
C06151=1046.513,186.242,-95.084,171.020,37.467,157.063
C06152=1046.507,185.994,-95.059,171.018,37.465,157.063
C06153=1046.501,185.745,-95.035,171.015,37.463,157.063
C06154=1046.495,185.496,-95.011,171.013,37.461,157.062
C06155=1046.489,185.247,-94.987,171.010,37.459,157.062
C06156=1046.484,184.998,-94.964,171.008,37.457,157.061
C06157=1046.478,184.750,-94.940,171.006,37.455,157.061
C06158=1046.472,184.501,-94.915,171.003,37.453,157.061
C06159=1046.466,184.252,-94.892,171.001,37.451,157.060
C06160=1046.460,184.003,-94.867,170.998,37.449,157.060
C06161=1046.454,183.755,-94.843,170.995,37.447,157.059
C06162=1046.448,183.506,-94.820,170.993,37.446,157.059
C06163=1046.441,183.257,-94.796,170.991,37.444,157.059
C06164=1046.435,183.009,-94.773,170.989,37.442,157.058
C06165=1046.429,182.759,-94.749,170.986,37.440,157.058
C06166=1046.423,182.511,-94.726,170.983,37.438,157.057
C06167=1046.416,182.262,-94.702,170.981,37.437,157.057
C06168=1046.410,182.013,-94.679,170.978,37.435,157.057
C06169=1046.403,181.764,-94.655,170.976,37.433,157.056
C06170=1046.397,181.516,-94.632,170.974,37.431,157.056
C06171=1046.391,181.266,-94.608,170.972,37.429,157.055
C06172=1046.385,181.018,-94.585,170.968,37.428,157.055
C06173=1046.379,180.768,-94.561,170.966,37.426,157.055
C06174=1046.372,180.520,-94.538,170.964,37.424,157.054
C06175=1046.366,180.271,-94.514,170.961,37.422,157.054
C06176=1046.360,180.022,-94.491,170.959,37.421,157.054
C06177=1046.354,179.774,-94.467,170.957,37.419,157.053
C06178=1046.348,179.524,-94.444,170.954,37.417,157.053
C06179=1046.342,179.276,-94.420,170.951,37.415,157.052
C06180=1046.335,179.026,-94.397,170.949,37.413,157.052
C06181=1046.329,178.779,-94.374,170.947,37.412,157.052
C06182=1046.323,178.530,-94.351,170.945,37.410,157.051
C06183=1046.316,178.281,-94.327,170.942,37.408,157.051
C06184=1046.311,178.032,-94.304,170.940,37.406,157.050
C06185=1046.304,177.783,-94.280,170.938,37.404,157.050
C06186=1046.298,177.534,-94.257,170.934,37.403,157.050
C06187=1046.292,177.286,-94.233,170.932,37.401,157.049
C06188=1046.286,177.036,-94.210,170.930,37.400,157.049
C06189=1046.280,176.788,-94.186,170.928,37.398,157.049
C06190=1046.274,176.539,-94.163,170.925,37.396,157.048
C06191=1046.267,176.290,-94.141,170.923,37.394,157.048
C06192=1046.261,176.041,-94.117,170.921,37.392,157.048
C06193=1046.255,175.792,-94.094,170.919,37.391,157.047
C06194=1046.249,175.543,-94.070,170.916,37.389,157.047
C06195=1046.243,175.294,-94.047,170.913,37.387,157.046
C06196=1046.237,175.046,-94.024,170.911,37.385,157.046
C06197=1046.231,174.797,-94.000,170.908,37.383,157.046
C06198=1046.225,174.548,-93.977,170.906,37.382,157.045
C06199=1046.219,174.299,-93.954,170.904,37.380,157.045
C06200=1046.213,174.083,-93.934,170.902,37.379,157.045
C06201=1046.209,173.869,-93.914,170.900,37.377,157.044
C06202=1046.202,173.654,-93.894,170.898,37.376,157.044
C06203=1046.197,173.438,-93.874,170.896,37.374,157.044
C06204=1046.192,173.224,-93.854,170.894,37.373,157.043
C06205=1046.187,173.008,-93.834,170.892,37.371,157.043
C06206=1046.181,172.793,-93.814,170.890,37.370,157.043
C06207=1046.176,172.578,-93.794,170.888,37.368,157.042
C06208=1046.171,172.329,-93.771,170.886,37.366,157.042
C06209=1046.164,172.080,-93.748,170.884,37.364,157.042
C06210=1046.158,171.831,-93.724,170.881,37.363,157.041
C06211=1046.152,171.582,-93.701,170.879,37.361,157.041
C06212=1046.147,171.334,-93.678,170.877,37.359,157.040
C06213=1046.140,171.085,-93.656,170.873,37.357,157.040
C06214=1046.134,170.836,-93.632,170.871,37.356,157.040
C06215=1046.128,170.587,-93.609,170.869,37.354,157.039
C06216=1046.122,170.338,-93.586,170.867,37.352,157.039
C06217=1046.116,170.089,-93.563,170.864,37.351,157.039
C06218=1046.111,169.840,-93.540,170.862,37.349,157.038
C06219=1046.104,169.591,-93.516,170.860,37.347,157.038
C06220=1046.098,169.343,-93.494,170.858,37.345,157.037
C06221=1046.092,169.094,-93.471,170.855,37.343,157.037
C06222=1046.086,168.845,-93.448,170.853,37.342,157.037
C06223=1046.080,168.596,-93.425,170.851,37.340,157.036
C06224=1046.075,168.347,-93.402,170.849,37.338,157.036
C06225=1046.069,168.098,-93.379,170.846,37.337,157.036
C06226=1046.062,167.849,-93.356,170.844,37.335,157.035
C06227=1046.056,167.601,-93.333,170.842,37.333,157.035
C06228=1046.050,167.352,-93.310,170.840,37.331,157.035
C06229=1046.044,167.103,-93.287,170.837,37.330,157.034
C06230=1046.039,166.854,-93.264,170.835,37.328,157.034
C06231=1046.032,166.606,-93.241,170.833,37.326,157.033
C06232=1046.026,166.357,-93.218,170.830,37.324,157.033
C06233=1046.021,166.108,-93.195,170.828,37.322,157.033
C06234=1046.015,165.859,-93.172,170.826,37.320,157.032
C06235=1046.009,165.610,-93.150,170.824,37.319,157.032
C06236=1046.002,165.361,-93.127,170.821,37.317,157.032
C06237=1045.996,165.112,-93.104,170.819,37.316,157.031
C06238=1045.991,164.863,-93.081,170.817,37.314,157.031
C06239=1045.985,164.614,-93.058,170.815,37.312,157.030
C06240=1045.977,164.262,-93.026,170.811,37.310,157.030
C06241=1045.968,163.910,-92.994,170.809,37.307,157.029
C06242=1045.960,163.558,-92.961,170.806,37.305,157.029
C06243=1045.952,163.205,-92.929,170.802,37.302,157.028
C06244=1045.946,162.956,-92.906,170.800,37.301,157.028
C06245=1045.940,162.707,-92.884,170.798,37.299,157.028
C06246=1045.934,162.458,-92.861,170.795,37.297,157.027
C06247=1045.928,162.210,-92.838,170.793,37.295,157.027
C06248=1045.922,161.961,-92.815,170.791,37.293,157.027
C06249=1045.917,161.712,-92.792,170.789,37.292,157.026
C06250=1045.910,161.463,-92.770,170.786,37.290,157.026
C06251=1045.905,161.214,-92.748,170.784,37.288,157.025
C06252=1045.899,160.965,-92.725,170.782,37.286,157.025
C06253=1045.893,160.716,-92.702,170.780,37.285,157.025
C06254=1045.887,160.467,-92.679,170.778,37.283,157.024
C06255=1045.881,160.218,-92.656,170.776,37.281,157.024
C06256=1045.875,159.969,-92.635,170.774,37.280,157.024
C06257=1045.869,159.720,-92.612,170.772,37.278,157.023
C06258=1045.863,159.472,-92.590,170.769,37.277,157.023
C06259=1045.857,159.222,-92.568,170.767,37.275,157.023
C06260=1045.851,158.974,-92.545,170.765,37.273,157.022
C06261=1045.844,158.725,-92.523,170.763,37.272,157.022
C06262=1045.839,158.475,-92.500,170.760,37.270,157.022
C06263=1045.833,158.227,-92.478,170.758,37.269,157.021
C06264=1045.825,157.941,-92.453,170.756,37.266,157.021
C06265=1045.819,157.657,-92.427,170.753,37.264,157.020
C06266=1045.811,157.371,-92.402,170.750,37.263,157.020
C06267=1045.805,157.085,-92.375,170.748,37.261,157.020
C06268=1045.798,156.836,-92.353,170.746,37.260,157.019
C06269=1045.792,156.588,-92.331,170.744,37.258,157.019
C06270=1045.786,156.339,-92.308,170.741,37.256,157.019
C06271=1045.781,156.090,-92.287,170.739,37.255,157.018
C06272=1045.774,155.842,-92.264,170.737,37.253,157.018
C06273=1045.769,155.592,-92.242,170.735,37.251,157.018
C06274=1045.762,155.343,-92.220,170.732,37.250,157.017
C06275=1045.756,155.094,-92.198,170.730,37.248,157.017
C06276=1045.750,154.845,-92.175,170.728,37.246,157.017
C06277=1045.744,154.596,-92.154,170.726,37.245,157.016
C06278=1045.738,154.348,-92.131,170.724,37.243,157.016
C06279=1045.732,154.098,-92.109,170.722,37.242,157.016
C06280=1045.726,153.849,-92.087,170.720,37.240,157.015
C06281=1045.720,153.600,-92.065,170.718,37.239,157.015
C06282=1045.713,153.352,-92.043,170.715,37.237,157.015
C06283=1045.708,153.102,-92.021,170.713,37.235,157.014
C06284=1045.701,152.854,-91.998,170.711,37.234,157.014
C06285=1045.695,152.604,-91.977,170.709,37.232,157.014
C06286=1045.689,152.356,-91.954,170.707,37.231,157.013
C06287=1045.683,152.107,-91.933,170.704,37.229,157.013
C06288=1045.678,151.858,-91.911,170.702,37.228,157.013
C06289=1045.671,151.609,-91.888,170.700,37.226,157.012
C06290=1045.665,151.360,-91.867,170.698,37.225,157.012
C06291=1045.659,151.111,-91.844,170.696,37.223,157.012
C06292=1045.653,150.862,-91.822,170.694,37.221,157.011
C06293=1045.647,150.613,-91.800,170.692,37.220,157.011
C06294=1045.641,150.364,-91.778,170.690,37.218,157.011
C06295=1045.634,150.115,-91.757,170.688,37.217,157.011
C06296=1045.629,149.866,-91.735,170.685,37.215,157.010
C06297=1045.623,149.617,-91.712,170.683,37.213,157.010
C06298=1045.617,149.368,-91.691,170.681,37.212,157.010
C06299=1045.611,149.119,-91.669,170.679,37.210,157.009
C06300=1045.604,148.870,-91.647,170.676,37.209,157.009
C06301=1045.598,148.621,-91.625,170.675,37.207,157.009
C06302=1045.592,148.372,-91.603,170.673,37.205,157.008
C06303=1045.586,148.124,-91.582,170.671,37.204,157.008
C06304=1045.580,147.875,-91.560,170.668,37.202,157.008
C06305=1045.575,147.625,-91.538,170.666,37.201,157.007
C06306=1045.568,147.376,-91.516,170.664,37.199,157.007
C06307=1045.562,147.127,-91.494,170.662,37.198,157.007
C06308=1045.556,146.878,-91.473,170.660,37.196,157.006
C06309=1045.550,146.629,-91.450,170.657,37.195,157.006
C06310=1045.544,146.381,-91.429,170.655,37.193,157.006
C06311=1045.538,146.132,-91.407,170.654,37.192,157.005
C06312=1045.532,145.882,-91.386,170.652,37.190,157.005
C06313=1045.526,145.633,-91.364,170.650,37.189,157.005
C06314=1045.519,145.384,-91.342,170.647,37.187,157.004
C06315=1045.513,145.135,-91.320,170.645,37.186,157.004
C06316=1045.507,144.887,-91.299,170.643,37.184,157.004
C06317=1045.500,144.638,-91.278,170.641,37.183,157.004
C06318=1045.494,144.389,-91.256,170.638,37.181,157.003
C06319=1045.488,144.140,-91.235,170.637,37.180,157.003
C06320=1045.482,143.890,-91.213,170.635,37.178,157.003
C06321=1045.476,143.642,-91.192,170.633,37.177,157.002
C06322=1045.470,143.393,-91.170,170.631,37.175,157.002
C06323=1045.464,143.143,-91.148,170.628,37.174,157.002
C06324=1045.458,142.894,-91.127,170.626,37.172,157.001
C06325=1045.452,142.646,-91.105,170.624,37.171,157.001
C06326=1045.446,142.397,-91.084,170.622,37.169,157.001
C06327=1045.440,142.147,-91.062,170.621,37.168,157.000
C06328=1045.433,141.862,-91.037,170.617,37.166,157.000
C06329=1045.426,141.577,-91.012,170.615,37.164,157.000
C06330=1045.419,141.291,-90.988,170.613,37.162,156.999
C06331=1045.412,141.005,-90.963,170.610,37.160,156.999
C06332=1045.406,140.756,-90.941,170.608,37.159,156.999
C06333=1045.400,140.508,-90.920,170.606,37.157,156.998
C06334=1045.393,140.259,-90.899,170.605,37.156,156.998
C06335=1045.387,140.009,-90.877,170.603,37.154,156.998
C06336=1045.382,139.760,-90.857,170.600,37.153,156.997
C06337=1045.376,139.511,-90.835,170.598,37.151,156.997
C06338=1045.370,139.262,-90.814,170.596,37.150,156.997
C06339=1045.364,139.013,-90.792,170.594,37.148,156.996
C06340=1045.358,138.764,-90.771,170.593,37.147,156.996
C06341=1045.351,138.515,-90.750,170.590,37.146,156.996
C06342=1045.345,138.266,-90.728,170.588,37.144,156.996
C06343=1045.339,138.017,-90.706,170.586,37.143,156.995
C06344=1045.333,137.768,-90.686,170.584,37.141,156.995
C06345=1045.327,137.519,-90.665,170.582,37.140,156.995
C06346=1045.320,137.270,-90.643,170.579,37.138,156.994
C06347=1045.315,137.021,-90.622,170.578,37.137,156.994
C06348=1045.309,136.772,-90.600,170.576,37.136,156.994
C06349=1045.302,136.523,-90.579,170.574,37.134,156.993
C06350=1045.297,136.274,-90.559,170.572,37.132,156.993
C06351=1045.290,136.025,-90.537,170.569,37.131,156.993
C06352=1045.283,135.776,-90.516,170.567,37.129,156.993
C06353=1045.278,135.527,-90.495,170.566,37.128,156.992
C06354=1045.272,135.277,-90.474,170.564,37.126,156.992
C06355=1045.265,135.029,-90.453,170.561,37.125,156.992
C06356=1045.260,134.780,-90.431,170.559,37.123,156.991
C06357=1045.253,134.531,-90.410,170.557,37.122,156.991
C06358=1045.247,134.281,-90.389,170.556,37.121,156.991
C06359=1045.241,134.033,-90.368,170.554,37.119,156.990
C06360=1045.235,133.784,-90.347,170.551,37.118,156.990
C06361=1045.229,133.534,-90.326,170.549,37.116,156.990
C06362=1045.223,133.286,-90.305,170.547,37.115,156.990
C06363=1045.217,133.036,-90.283,170.545,37.114,156.989
C06364=1045.211,132.788,-90.263,170.544,37.112,156.989
C06365=1045.205,132.538,-90.242,170.541,37.111,156.989
C06366=1045.198,132.289,-90.220,170.539,37.109,156.988
C06367=1045.192,132.040,-90.200,170.537,37.108,156.988
C06368=1045.186,131.791,-90.178,170.535,37.106,156.988
C06369=1045.180,131.542,-90.157,170.534,37.104,156.987
C06370=1045.174,131.293,-90.137,170.531,37.103,156.987
C06371=1045.168,131.044,-90.115,170.529,37.101,156.987
C06372=1045.162,130.795,-90.095,170.527,37.100,156.987
C06373=1045.156,130.546,-90.074,170.525,37.099,156.986
C06374=1045.149,130.296,-90.053,170.523,37.098,156.986
C06375=1045.143,130.048,-90.033,170.521,37.096,156.986
C06376=1045.137,129.798,-90.012,170.519,37.095,156.985
C06377=1045.130,129.550,-89.991,170.517,37.094,156.985
C06378=1045.125,129.300,-89.970,170.515,37.092,156.985
C06379=1045.118,129.052,-89.949,170.513,37.090,156.985
C06380=1045.112,128.803,-89.929,170.511,37.089,156.984
C06381=1045.106,128.553,-89.907,170.509,37.088,156.984
C06382=1045.099,128.304,-89.887,170.507,37.087,156.984
C06383=1045.093,128.056,-89.866,170.505,37.085,156.983
C06384=1045.087,127.806,-89.846,170.503,37.084,156.983
C06385=1045.081,127.558,-89.825,170.502,37.083,156.983
C06386=1045.074,127.308,-89.805,170.499,37.081,156.983
C06387=1045.068,127.058,-89.784,170.497,37.080,156.982
C06388=1045.062,126.810,-89.763,170.495,37.078,156.982
C06389=1045.055,126.561,-89.743,170.493,37.077,156.982
C06390=1045.050,126.312,-89.721,170.492,37.075,156.981
C06391=1045.043,126.063,-89.701,170.489,37.074,156.981
C06392=1045.036,125.777,-89.677,170.487,37.073,156.981
C06393=1045.029,125.491,-89.653,170.485,37.071,156.981
C06394=1045.022,125.205,-89.630,170.483,37.069,156.980
C06395=1045.016,124.919,-89.606,170.481,37.068,156.980
C06396=1045.009,124.670,-89.586,170.478,37.066,156.980
C06397=1045.003,124.422,-89.565,170.476,37.065,156.979
C06398=1044.997,124.172,-89.544,170.474,37.064,156.979
C06399=1044.991,123.923,-89.524,170.472,37.062,156.979
C06400=1044.984,123.674,-89.503,170.471,37.061,156.978
C06401=1044.979,123.425,-89.483,170.468,37.059,156.978
C06402=1044.972,123.176,-89.462,170.466,37.058,156.978
C06403=1044.966,122.927,-89.442,170.464,37.056,156.978
C06404=1044.960,122.678,-89.421,170.462,37.055,156.977
C06405=1044.954,122.429,-89.401,170.461,37.054,156.977
C06406=1044.948,122.179,-89.381,170.458,37.053,156.977
C06407=1044.941,121.931,-89.360,170.456,37.051,156.976
C06408=1044.935,121.681,-89.339,170.454,37.050,156.976
C06409=1044.929,121.432,-89.319,170.453,37.048,156.976
C06410=1044.923,121.183,-89.299,170.451,37.047,156.976
C06411=1044.917,120.934,-89.277,170.448,37.045,156.975
C06412=1044.911,120.685,-89.257,170.446,37.044,156.975
C06413=1044.905,120.436,-89.237,170.445,37.042,156.975
C06414=1044.899,120.187,-89.217,170.443,37.041,156.975
C06415=1044.893,119.937,-89.196,170.441,37.040,156.974
C06416=1044.886,119.689,-89.176,170.438,37.038,156.974
C06417=1044.881,119.439,-89.155,170.437,37.037,156.974
C06418=1044.875,119.191,-89.135,170.435,37.036,156.973
C06419=1044.869,118.942,-89.115,170.433,37.034,156.973
C06420=1044.862,118.692,-89.094,170.431,37.032,156.973
C06421=1044.857,118.443,-89.074,170.429,37.031,156.973
C06422=1044.850,118.194,-89.053,170.427,37.030,156.972
C06423=1044.844,117.945,-89.033,170.425,37.028,156.972
C06424=1044.839,117.696,-89.012,170.423,37.027,156.972
C06425=1044.832,117.447,-88.992,170.422,37.026,156.971
C06426=1044.826,117.198,-88.972,170.419,37.024,156.971
C06427=1044.819,116.948,-88.952,170.417,37.023,156.971
C06428=1044.814,116.699,-88.931,170.415,37.021,156.971
C06429=1044.808,116.451,-88.911,170.414,37.020,156.970
C06430=1044.802,116.201,-88.891,170.412,37.018,156.970
C06431=1044.796,115.952,-88.870,170.410,37.017,156.970
C06432=1044.790,115.704,-88.850,170.408,37.015,156.969
C06433=1044.783,115.454,-88.829,170.406,37.014,156.969
C06434=1044.777,115.205,-88.809,170.404,37.013,156.969
C06435=1044.772,114.956,-88.789,170.402,37.011,156.968
C06436=1044.766,114.707,-88.768,170.401,37.010,156.968
C06437=1044.760,114.458,-88.748,170.398,37.009,156.968
C06438=1044.754,114.209,-88.729,170.396,37.007,156.968
C06439=1044.748,113.959,-88.708,170.394,37.005,156.967
C06440=1044.742,113.710,-88.688,170.393,37.004,156.967
C06441=1044.736,113.462,-88.668,170.391,37.002,156.967
C06442=1044.729,113.212,-88.647,170.388,37.001,156.966
C06443=1044.723,112.963,-88.627,170.387,37.000,156.966
C06444=1044.717,112.714,-88.608,170.385,36.999,156.966
C06445=1044.711,112.464,-88.588,170.383,36.998,156.966
C06446=1044.705,112.216,-88.568,170.381,36.996,156.965
C06447=1044.699,111.967,-88.548,170.380,36.994,156.965
C06448=1044.692,111.717,-88.528,170.377,36.993,156.965
C06449=1044.686,111.468,-88.508,170.375,36.992,156.965
C06450=1044.680,111.220,-88.488,170.373,36.991,156.964
C06451=1044.674,110.970,-88.467,170.372,36.989,156.964
C06452=1044.668,110.721,-88.448,170.370,36.988,156.964
C06453=1044.662,110.472,-88.428,170.367,36.986,156.964
C06454=1044.655,110.222,-88.408,170.365,36.985,156.963
C06455=1044.649,109.974,-88.388,170.364,36.984,156.963
C06456=1044.642,109.688,-88.365,170.362,36.982,156.963
C06457=1044.635,109.402,-88.343,170.360,36.981,156.962
C06458=1044.628,109.115,-88.319,170.357,36.979,156.962
C06459=1044.621,108.829,-88.297,170.355,36.978,156.962
C06460=1044.615,108.581,-88.277,170.353,36.977,156.962
C06461=1044.609,108.332,-88.257,170.351,36.975,156.961
C06462=1044.602,108.082,-88.237,170.349,36.974,156.961
C06463=1044.596,107.833,-88.218,170.348,36.972,156.961
C06464=1044.590,107.584,-88.198,170.345,36.971,156.960
C06465=1044.584,107.336,-88.178,170.343,36.970,156.960
C06466=1044.577,107.085,-88.158,170.342,36.969,156.960
C06467=1044.571,106.837,-88.139,170.340,36.967,156.960
C06468=1044.565,106.588,-88.119,170.338,36.966,156.959
C06469=1044.559,106.338,-88.099,170.336,36.964,156.959
C06470=1044.552,106.089,-88.080,170.334,36.963,156.959
C06471=1044.546,105.840,-88.060,170.332,36.962,156.959
C06472=1044.541,105.591,-88.040,170.330,36.961,156.958
C06473=1044.534,105.341,-88.020,170.329,36.959,156.958
C06474=1044.528,105.093,-88.000,170.327,36.958,156.958
C06475=1044.522,104.843,-87.981,170.324,36.956,156.958
C06476=1044.516,104.595,-87.962,170.322,36.955,156.957
C06477=1044.510,104.346,-87.942,170.321,36.954,156.957
C06478=1044.503,104.096,-87.922,170.319,36.953,156.957
C06479=1044.497,103.847,-87.902,170.317,36.951,156.957
C06480=1044.492,103.597,-87.883,170.316,36.950,156.956
C06481=1044.485,103.349,-87.863,170.313,36.948,156.956
C06482=1044.478,103.099,-87.843,170.311,36.947,156.956
C06483=1044.473,102.850,-87.824,170.309,36.946,156.955
C06484=1044.467,102.601,-87.804,170.308,36.945,156.955
C06485=1044.461,102.352,-87.785,170.306,36.943,156.955
C06486=1044.455,102.103,-87.765,170.304,36.942,156.955
C06487=1044.448,101.854,-87.746,170.302,36.940,156.954
C06488=1044.442,101.604,-87.726,170.300,36.939,156.954
C06489=1044.436,101.355,-87.706,170.298,36.938,156.954
C06490=1044.430,101.106,-87.686,170.296,36.937,156.954
C06491=1044.424,100.857,-87.667,170.295,36.935,156.953
C06492=1044.418,100.608,-87.648,170.292,36.934,156.953
C06493=1044.412,100.359,-87.629,170.290,36.932,156.953
C06494=1044.406,100.109,-87.608,170.289,36.931,156.952
C06495=1044.399,99.860,-87.590,170.287,36.930,156.952
C06496=1044.393,99.611,-87.570,170.285,36.929,156.952
C06497=1044.387,99.362,-87.551,170.283,36.927,156.952
C06498=1044.381,99.113,-87.531,170.282,36.926,156.952
C06499=1044.374,98.863,-87.512,170.279,36.925,156.951
C06500=1044.368,98.614,-87.493,170.277,36.924,156.951
C06501=1044.362,98.365,-87.473,170.276,36.922,156.951
C06502=1044.356,98.116,-87.454,170.274,36.921,156.950
C06503=1044.350,97.867,-87.434,170.272,36.919,156.950
C06504=1044.343,97.617,-87.415,170.269,36.918,156.950
C06505=1044.337,97.368,-87.396,170.268,36.917,156.950
C06506=1044.330,97.120,-87.377,170.266,36.916,156.949
C06507=1044.324,96.870,-87.357,170.264,36.914,156.949
C06508=1044.318,96.621,-87.339,170.263,36.913,156.949
C06509=1044.312,96.372,-87.319,170.261,36.912,156.949
C06510=1044.306,96.123,-87.300,170.258,36.911,156.948
C06511=1044.300,95.874,-87.281,170.257,36.910,156.948
C06512=1044.293,95.624,-87.261,170.255,36.908,156.948
C06513=1044.287,95.375,-87.242,170.253,36.906,156.948
C06514=1044.281,95.126,-87.223,170.251,36.905,156.947
C06515=1044.274,94.877,-87.203,170.250,36.904,156.947
C06516=1044.269,94.628,-87.184,170.247,36.903,156.947
C06517=1044.262,94.378,-87.165,170.245,36.902,156.947
C06518=1044.257,94.129,-87.146,170.244,36.900,156.946
C06519=1044.250,93.881,-87.127,170.242,36.899,156.946
C06520=1044.243,93.594,-87.105,170.240,36.897,156.946
C06521=1044.236,93.308,-87.082,170.238,36.896,156.946
C06522=1044.229,93.022,-87.061,170.235,36.895,156.945
C06523=1044.222,92.736,-87.039,170.233,36.893,156.945
C06524=1044.215,92.487,-87.020,170.231,36.892,156.945
C06525=1044.209,92.238,-87.000,170.230,36.890,156.944
C06526=1044.203,91.988,-86.982,170.228,36.889,156.944
C06527=1044.197,91.739,-86.962,170.226,36.888,156.944
C06528=1044.192,91.490,-86.943,170.224,36.886,156.944
C06529=1044.185,91.241,-86.924,170.222,36.885,156.943
C06530=1044.179,90.992,-86.905,170.220,36.884,156.943
C06531=1044.173,90.743,-86.886,170.219,36.882,156.943
C06532=1044.167,90.493,-86.867,170.217,36.881,156.943
C06533=1044.161,90.244,-86.848,170.215,36.880,156.942
C06534=1044.154,89.995,-86.829,170.213,36.879,156.942
C06535=1044.149,89.745,-86.810,170.211,36.877,156.942
C06536=1044.142,89.496,-86.792,170.209,36.876,156.942
C06537=1044.135,89.248,-86.772,170.207,36.875,156.941
C06538=1044.129,88.999,-86.754,170.206,36.874,156.941
C06539=1044.123,88.749,-86.734,170.204,36.872,156.941
C06540=1044.116,88.499,-86.715,170.201,36.871,156.941
C06541=1044.110,88.250,-86.697,170.200,36.870,156.940
C06542=1044.103,88.001,-86.678,170.198,36.869,156.940
C06543=1044.098,87.752,-86.659,170.196,36.868,156.940
C06544=1044.091,87.503,-86.640,170.194,36.866,156.940
C06545=1044.085,87.254,-86.621,170.193,36.865,156.939
C06546=1044.078,87.004,-86.603,170.190,36.864,156.939
C06547=1044.073,86.755,-86.584,170.188,36.863,156.939
C06548=1044.066,86.506,-86.565,170.187,36.861,156.939
C06549=1044.060,86.257,-86.546,170.185,36.860,156.938
C06550=1044.053,86.008,-86.528,170.183,36.859,156.938
C06551=1044.047,85.758,-86.509,170.182,36.858,156.938
C06552=1044.041,85.509,-86.490,170.180,36.856,156.938
C06553=1044.035,85.260,-86.471,170.177,36.855,156.937
C06554=1044.028,85.011,-86.452,170.175,36.854,156.937
C06555=1044.022,84.761,-86.434,170.174,36.853,156.937
C06556=1044.017,84.512,-86.415,170.172,36.851,156.937
C06557=1044.010,84.262,-86.397,170.170,36.850,156.937
C06558=1044.004,84.013,-86.378,170.169,36.849,156.936
C06559=1043.997,83.764,-86.359,170.166,36.848,156.936
C06560=1043.991,83.515,-86.341,170.164,36.846,156.936
C06561=1043.985,83.266,-86.321,170.163,36.845,156.936
C06562=1043.979,83.017,-86.303,170.161,36.844,156.935
C06563=1043.973,82.768,-86.284,170.159,36.843,156.935
C06564=1043.967,82.519,-86.266,170.158,36.841,156.935
C06565=1043.960,82.269,-86.248,170.155,36.840,156.934
C06566=1043.955,82.020,-86.229,170.153,36.838,156.934
C06567=1043.948,81.771,-86.210,170.152,36.837,156.934
C06568=1043.942,81.522,-86.191,170.150,36.836,156.934
C06569=1043.935,81.273,-86.173,170.148,36.835,156.933
C06570=1043.930,81.023,-86.153,170.146,36.833,156.933
C06571=1043.924,80.773,-86.136,170.144,36.832,156.933
C06572=1043.917,80.524,-86.117,170.142,36.831,156.933
C06573=1043.911,80.275,-86.098,170.140,36.830,156.933
C06574=1043.904,80.026,-86.080,170.139,36.828,156.932
C06575=1043.899,79.778,-86.061,170.137,36.827,156.932
C06576=1043.893,79.527,-86.043,170.135,36.826,156.932
C06577=1043.887,79.278,-86.024,170.134,36.825,156.932
C06578=1043.880,79.029,-86.005,170.131,36.823,156.931
C06579=1043.874,78.780,-85.987,170.129,36.822,156.931
C06580=1043.868,78.530,-85.969,170.128,36.821,156.931
C06581=1043.861,78.281,-85.950,170.126,36.820,156.931
C06582=1043.856,78.032,-85.931,170.124,36.819,156.930
C06583=1043.850,77.783,-85.913,170.123,36.817,156.930
C06584=1043.842,77.497,-85.892,170.120,36.815,156.930
C06585=1043.835,77.210,-85.871,170.118,36.814,156.929
C06586=1043.828,76.925,-85.850,170.116,36.813,156.929
C06587=1043.821,76.639,-85.828,170.114,36.812,156.929
C06588=1043.815,76.389,-85.811,170.112,36.810,156.929
C06589=1043.808,76.140,-85.792,170.110,36.809,156.929
C06590=1043.802,75.891,-85.773,170.108,36.808,156.928
C06591=1043.796,75.642,-85.756,170.106,36.807,156.928
C06592=1043.789,75.393,-85.738,170.104,36.805,156.928
C06593=1043.783,75.143,-85.720,170.103,36.804,156.928
C06594=1043.777,74.894,-85.701,170.101,36.803,156.927
C06595=1043.770,74.645,-85.682,170.099,36.802,156.927
C06596=1043.764,74.395,-85.664,170.097,36.801,156.927
C06597=1043.758,74.147,-85.646,170.095,36.799,156.927
C06598=1043.752,73.897,-85.628,170.093,36.798,156.926
C06599=1043.746,73.648,-85.610,170.091,36.797,156.926
C06600=1043.740,73.398,-85.592,170.090,36.796,156.926
C06601=1043.733,73.149,-85.573,170.088,36.794,156.926
C06602=1043.727,72.899,-85.555,170.086,36.793,156.925
C06603=1043.721,72.651,-85.537,170.084,36.792,156.925
C06604=1043.715,72.402,-85.518,170.082,36.791,156.925
C06605=1043.709,72.152,-85.500,170.080,36.789,156.925
C06606=1043.701,71.903,-85.482,170.079,36.788,156.924
C06607=1043.695,71.654,-85.464,170.077,36.787,156.924
C06608=1043.690,71.404,-85.447,170.075,36.786,156.924
C06609=1043.683,71.155,-85.428,170.073,36.784,156.924
C06610=1043.677,70.906,-85.410,170.071,36.783,156.923
C06611=1043.671,70.656,-85.391,170.069,36.782,156.923
C06612=1043.665,70.407,-85.373,170.067,36.781,156.923
C06613=1043.659,70.158,-85.355,170.066,36.780,156.923
C06614=1043.652,69.909,-85.338,170.064,36.779,156.923
C06615=1043.646,69.660,-85.319,170.062,36.777,156.922
C06616=1043.639,69.410,-85.301,170.060,36.776,156.922
C06617=1043.634,69.161,-85.284,170.058,36.775,156.922
C06618=1043.628,68.912,-85.265,170.056,36.774,156.922
C06619=1043.621,68.662,-85.248,170.055,36.772,156.921
C06620=1043.614,68.413,-85.229,170.053,36.771,156.921
C06621=1043.608,68.164,-85.211,170.051,36.770,156.921
C06622=1043.603,67.915,-85.194,170.049,36.769,156.921
C06623=1043.595,67.666,-85.176,170.047,36.768,156.920
C06624=1043.589,67.416,-85.158,170.045,36.766,156.920
C06625=1043.583,67.166,-85.140,170.043,36.765,156.920
C06626=1043.577,66.918,-85.121,170.042,36.764,156.920
C06627=1043.571,66.668,-85.104,170.040,36.763,156.920
C06628=1043.564,66.419,-85.086,170.038,36.762,156.919
C06629=1043.558,66.170,-85.067,170.037,36.761,156.919
C06630=1043.552,65.921,-85.050,170.034,36.759,156.919
C06631=1043.546,65.671,-85.033,170.032,36.758,156.919
C06632=1043.539,65.421,-85.015,170.030,36.757,156.918
C06633=1043.534,65.173,-84.996,170.029,36.756,156.918
C06634=1043.527,64.923,-84.979,170.027,36.754,156.918
C06635=1043.521,64.674,-84.961,170.025,36.753,156.918
C06636=1043.515,64.424,-84.943,170.024,36.752,156.917
C06637=1043.508,64.176,-84.925,170.021,36.751,156.917
C06638=1043.502,63.926,-84.908,170.019,36.750,156.917
C06639=1043.495,63.677,-84.890,170.018,36.749,156.917
C06640=1043.489,63.427,-84.872,170.016,36.748,156.917
C06641=1043.483,63.178,-84.855,170.014,36.746,156.916
C06642=1043.477,62.928,-84.837,170.012,36.745,156.916
C06643=1043.469,62.680,-84.819,170.011,36.744,156.916
C06644=1043.463,62.430,-84.801,170.008,36.743,156.916
C06645=1043.457,62.181,-84.784,170.006,36.742,156.916
C06646=1043.451,61.931,-84.766,170.004,36.741,156.915
C06647=1043.444,61.682,-84.749,170.003,36.740,156.915
C06648=1043.437,61.396,-84.729,170.001,36.738,156.915
C06649=1043.429,61.109,-84.709,169.999,36.737,156.915
C06650=1043.423,60.824,-84.689,169.997,36.736,156.914
C06651=1043.415,60.537,-84.669,169.994,36.734,156.914
C06652=1043.409,60.288,-84.652,169.992,36.734,156.914
C06653=1043.402,60.039,-84.634,169.990,36.733,156.914
C06654=1043.395,59.790,-84.616,169.989,36.731,156.913
C06655=1043.389,59.540,-84.598,169.987,36.730,156.913
C06656=1043.383,59.291,-84.581,169.985,36.729,156.913
C06657=1043.376,59.042,-84.563,169.983,36.728,156.913
C06658=1043.370,58.792,-84.545,169.981,36.727,156.913
C06659=1043.364,58.543,-84.528,169.979,36.726,156.912
C06660=1043.357,58.294,-84.511,169.977,36.724,156.912
C06661=1043.351,58.045,-84.494,169.975,36.723,156.912
C06662=1043.345,57.795,-84.476,169.974,36.723,156.912
C06663=1043.338,57.546,-84.458,169.972,36.721,156.912
C06664=1043.332,57.297,-84.441,169.970,36.720,156.911
C06665=1043.325,57.047,-84.424,169.969,36.719,156.911
C06666=1043.319,56.798,-84.406,169.966,36.718,156.911
C06667=1043.313,56.549,-84.389,169.964,36.717,156.911
C06668=1043.306,56.300,-84.372,169.962,36.716,156.910
C06669=1043.300,56.049,-84.355,169.961,36.714,156.910
C06670=1043.294,55.800,-84.338,169.959,36.713,156.910
C06671=1043.288,55.551,-84.320,169.957,36.712,156.910
C06672=1043.282,55.302,-84.303,169.956,36.711,156.910
C06673=1043.275,55.053,-84.285,169.953,36.710,156.909
C06674=1043.269,54.803,-84.267,169.951,36.709,156.909
C06675=1043.262,54.554,-84.250,169.949,36.708,156.909
C06676=1043.256,54.304,-84.232,169.948,36.706,156.909
C06677=1043.250,54.056,-84.215,169.946,36.705,156.908
C06678=1043.243,53.806,-84.198,169.944,36.704,156.908
C06679=1043.238,53.557,-84.181,169.942,36.703,156.908
C06680=1043.231,53.307,-84.164,169.940,36.702,156.908
C06681=1043.224,53.058,-84.147,169.938,36.701,156.908
C06682=1043.219,52.809,-84.129,169.936,36.699,156.907
C06683=1043.212,52.559,-84.112,169.935,36.698,156.907
C06684=1043.206,52.310,-84.095,169.933,36.697,156.907
C06685=1043.199,52.061,-84.077,169.931,36.696,156.907
C06686=1043.194,51.811,-84.061,169.929,36.695,156.907
C06687=1043.187,51.562,-84.043,169.928,36.694,156.906
C06688=1043.181,51.313,-84.026,169.925,36.693,156.906
C06689=1043.174,51.063,-84.008,169.923,36.691,156.906
C06690=1043.169,50.814,-83.991,169.922,36.690,156.906
C06691=1043.162,50.564,-83.974,169.920,36.689,156.905
C06692=1043.156,50.316,-83.957,169.918,36.688,156.905
C06693=1043.150,50.066,-83.939,169.916,36.687,156.905
C06694=1043.144,49.817,-83.922,169.915,36.686,156.905
C06695=1043.137,49.568,-83.905,169.912,36.684,156.905
C06696=1043.132,49.318,-83.888,169.910,36.683,156.904
C06697=1043.125,49.069,-83.871,169.909,36.682,156.904
C06698=1043.118,48.820,-83.854,169.907,36.681,156.904
C06699=1043.113,48.570,-83.837,169.905,36.680,156.904
C06700=1043.106,48.321,-83.820,169.903,36.679,156.903
C06701=1043.099,48.071,-83.802,169.902,36.677,156.903
C06702=1043.094,47.822,-83.785,169.899,36.676,156.903
C06703=1043.087,47.572,-83.768,169.897,36.675,156.903
C06704=1043.081,47.324,-83.751,169.896,36.674,156.902
C06705=1043.076,47.075,-83.733,169.894,36.672,156.902
C06706=1043.069,46.825,-83.717,169.892,36.671,156.902
C06707=1043.063,46.576,-83.700,169.890,36.671,156.902
C06708=1043.057,46.326,-83.682,169.889,36.669,156.902
C06709=1043.051,46.077,-83.666,169.886,36.668,156.901
C06710=1043.044,45.827,-83.648,169.884,36.667,156.901
C06711=1043.038,45.578,-83.631,169.882,36.666,156.901
C06712=1043.031,45.292,-83.612,169.881,36.664,156.901
C06713=1043.024,45.005,-83.593,169.879,36.663,156.900
C06714=1043.017,44.719,-83.573,169.877,36.661,156.900
C06715=1043.010,44.432,-83.553,169.875,36.660,156.900
C06716=1043.003,44.183,-83.536,169.872,36.659,156.900
C06717=1042.998,43.933,-83.519,169.870,36.658,156.900
C06718=1042.991,43.684,-83.502,169.868,36.657,156.899
C06719=1042.985,43.434,-83.486,169.867,36.656,156.899
C06720=1042.980,43.185,-83.468,169.865,36.654,156.899
C06721=1042.973,42.935,-83.451,169.863,36.653,156.899
C06722=1042.967,42.687,-83.434,169.861,36.652,156.898
C06723=1042.960,42.436,-83.418,169.859,36.651,156.898
C06724=1042.954,42.188,-83.401,169.857,36.650,156.898
C06725=1042.948,41.938,-83.385,169.855,36.649,156.898
C06726=1042.941,41.689,-83.367,169.853,36.647,156.897
C06727=1042.935,41.440,-83.351,169.852,36.647,156.897
C06728=1042.928,41.190,-83.334,169.850,36.645,156.897
C06729=1042.923,40.941,-83.317,169.848,36.644,156.897
C06730=1042.916,40.692,-83.300,169.846,36.643,156.897
C06731=1042.910,40.442,-83.284,169.844,36.642,156.897
C06732=1042.903,40.193,-83.267,169.842,36.641,156.896
C06733=1042.898,39.944,-83.251,169.840,36.640,156.896
C06734=1042.891,39.694,-83.234,169.839,36.639,156.896
C06735=1042.885,39.445,-83.217,169.837,36.637,156.896
C06736=1042.878,39.195,-83.200,169.835,36.637,156.895
C06737=1042.872,38.946,-83.183,169.833,36.635,156.895
C06738=1042.867,38.697,-83.167,169.832,36.634,156.895
C06739=1042.860,38.447,-83.150,169.829,36.633,156.895
C06740=1042.854,38.198,-83.133,169.827,36.632,156.895
C06741=1042.848,37.949,-83.117,169.825,36.631,156.894
C06742=1042.841,37.699,-83.100,169.824,36.630,156.894
C06743=1042.835,37.450,-83.083,169.822,36.628,156.894
C06744=1042.829,37.201,-83.067,169.820,36.628,156.894
C06745=1042.822,36.951,-83.051,169.818,36.627,156.894
C06746=1042.816,36.702,-83.034,169.815,36.625,156.893
C06747=1042.810,36.453,-83.018,169.814,36.625,156.893
C06748=1042.803,36.203,-83.001,169.812,36.623,156.893
C06749=1042.797,35.953,-82.985,169.810,36.622,156.893
C06750=1042.791,35.705,-82.968,169.808,36.622,156.893
C06751=1042.784,35.455,-82.952,169.807,36.620,156.892
C06752=1042.778,35.205,-82.935,169.805,36.619,156.892
C06753=1042.772,34.956,-82.919,169.803,36.618,156.892
C06754=1042.765,34.707,-82.902,169.801,36.617,156.892
C06755=1042.759,34.457,-82.886,169.798,36.616,156.892
C06756=1042.753,34.208,-82.869,169.797,36.615,156.891
C06757=1042.746,33.958,-82.853,169.795,36.614,156.891
C06758=1042.739,33.710,-82.836,169.793,36.613,156.891
C06759=1042.733,33.460,-82.820,169.791,36.611,156.891
C06760=1042.727,33.210,-82.803,169.790,36.611,156.891
C06761=1042.721,32.961,-82.787,169.788,36.610,156.890
C06762=1042.714,32.712,-82.772,169.786,36.608,156.890
C06763=1042.708,32.462,-82.755,169.783,36.608,156.890
C06764=1042.701,32.213,-82.738,169.781,36.606,156.890
C06765=1042.695,31.964,-82.722,169.780,36.605,156.890
C06766=1042.690,31.714,-82.705,169.778,36.605,156.889
C06767=1042.683,31.465,-82.690,169.776,36.603,156.889
C06768=1042.676,31.215,-82.673,169.774,36.602,156.889
C06769=1042.670,30.966,-82.657,169.772,36.601,156.889
C06770=1042.664,30.716,-82.641,169.771,36.600,156.889
C06771=1042.658,30.467,-82.624,169.768,36.599,156.888
C06772=1042.651,30.217,-82.608,169.766,36.598,156.888
C06773=1042.645,29.969,-82.591,169.764,36.597,156.888
C06774=1042.639,29.719,-82.575,169.763,36.596,156.888
C06775=1042.633,29.470,-82.559,169.761,36.594,156.888
C06776=1042.626,29.183,-82.541,169.759,36.593,156.887
C06777=1042.618,28.896,-82.522,169.757,36.593,156.887
C06778=1042.611,28.610,-82.503,169.755,36.591,156.887
C06779=1042.604,28.323,-82.484,169.752,36.590,156.887
C06780=1042.597,28.074,-82.468,169.750,36.589,156.886
C06781=1042.591,27.825,-82.452,169.748,36.587,156.886
C06782=1042.585,27.575,-82.435,169.746,36.587,156.886
C06783=1042.578,27.325,-82.421,169.744,36.586,156.886
C06784=1042.572,27.076,-82.404,169.743,36.585,156.886
C06785=1042.566,26.827,-82.388,169.741,36.584,156.886
C06786=1042.560,26.578,-82.372,169.739,36.582,156.885
C06787=1042.553,26.327,-82.356,169.737,36.582,156.885
C06788=1042.546,26.078,-82.340,169.734,36.581,156.885
C06789=1042.540,25.829,-82.324,169.733,36.580,156.885
C06790=1042.535,25.580,-82.308,169.731,36.579,156.885
C06791=1042.528,25.331,-82.292,169.729,36.577,156.884
C06792=1042.521,25.081,-82.275,169.727,36.577,156.884
C06793=1042.515,24.832,-82.260,169.725,36.575,156.884
C06794=1042.509,24.582,-82.243,169.723,36.575,156.884
C06795=1042.502,24.333,-82.228,169.722,36.574,156.884
C06796=1042.496,24.083,-82.212,169.719,36.572,156.883
C06797=1042.490,23.834,-82.196,169.717,36.572,156.883
C06798=1042.483,23.584,-82.180,169.715,36.570,156.883
C06799=1042.477,23.335,-82.164,169.713,36.570,156.883
C06800=1042.470,23.086,-82.148,169.712,36.568,156.883
C06801=1042.464,22.836,-82.132,169.710,36.567,156.882
C06802=1042.458,22.587,-82.117,169.708,36.567,156.882
C06803=1042.452,22.337,-82.101,169.706,36.565,156.882
C06804=1042.445,22.088,-82.085,169.704,36.565,156.882
C06805=1042.439,21.838,-82.068,169.701,36.563,156.882
C06806=1042.433,21.589,-82.052,169.700,36.562,156.882
C06807=1042.427,21.339,-82.037,169.698,36.562,156.881
C06808=1042.421,21.090,-82.021,169.696,36.560,156.881
C06809=1042.414,20.841,-82.005,169.694,36.560,156.881
C06810=1042.408,20.592,-81.989,169.692,36.558,156.881
C06811=1042.401,20.343,-81.973,169.691,36.557,156.881
C06812=1042.396,20.093,-81.958,169.689,36.556,156.880
C06813=1042.389,19.844,-81.942,169.687,36.555,156.880
C06814=1042.382,19.594,-81.925,169.684,36.555,156.880
C06815=1042.376,19.344,-81.910,169.682,36.553,156.880
C06816=1042.369,19.095,-81.895,169.680,36.552,156.880
C06817=1042.363,18.845,-81.878,169.678,36.551,156.880
C06818=1042.357,18.596,-81.864,169.677,36.550,156.879
C06819=1042.351,18.346,-81.847,169.675,36.549,156.879
C06820=1042.344,18.097,-81.832,169.673,36.548,156.879
C06821=1042.338,17.848,-81.817,169.671,36.548,156.879
C06822=1042.332,17.598,-81.800,169.669,36.546,156.879
C06823=1042.325,17.349,-81.785,169.666,36.546,156.878
C06824=1042.320,17.099,-81.769,169.665,36.544,156.878
C06825=1042.313,16.850,-81.754,169.663,36.544,156.878
C06826=1042.306,16.601,-81.738,169.661,36.543,156.878
C06827=1042.300,16.351,-81.722,169.659,36.541,156.878
C06828=1042.293,16.102,-81.706,169.657,36.541,156.878
C06829=1042.288,15.852,-81.691,169.655,36.539,156.877
C06830=1042.281,15.603,-81.675,169.654,36.539,156.877
C06831=1042.274,15.354,-81.659,169.652,36.537,156.877
C06832=1042.269,15.104,-81.644,169.649,36.537,156.877
C06833=1042.262,14.855,-81.628,169.647,36.536,156.877
C06834=1042.256,14.605,-81.613,169.645,36.535,156.876
C06835=1042.250,14.356,-81.597,169.643,36.534,156.876
C06836=1042.243,14.106,-81.582,169.641,36.532,156.876
C06837=1042.237,13.857,-81.566,169.640,36.532,156.876
C06838=1042.231,13.607,-81.551,169.638,36.531,156.876
C06839=1042.224,13.358,-81.535,169.636,36.530,156.876
C06840=1042.217,13.073,-81.518,169.634,36.529,156.875
C06841=1042.210,12.787,-81.501,169.631,36.528,156.875
C06842=1042.202,12.502,-81.483,169.628,36.527,156.875
C06843=1042.194,12.216,-81.465,169.626,36.526,156.875
C06844=1042.188,11.967,-81.450,169.624,36.525,156.875
C06845=1042.181,11.718,-81.435,169.622,36.524,156.875
C06846=1042.176,11.468,-81.419,169.620,36.523,156.874
C06847=1042.169,11.219,-81.403,169.619,36.522,156.874
C06848=1042.163,10.969,-81.388,169.617,36.522,156.874
C06849=1042.156,10.720,-81.373,169.615,36.520,156.874
C06850=1042.150,10.470,-81.358,169.613,36.520,156.874
C06851=1042.143,10.221,-81.343,169.610,36.518,156.873
C06852=1042.137,9.972,-81.327,169.608,36.518,156.873
C06853=1042.130,9.722,-81.312,169.606,36.517,156.873
C06854=1042.124,9.472,-81.297,169.604,36.516,156.873
C06855=1042.118,9.223,-81.281,169.602,36.515,156.873
C06856=1042.111,8.973,-81.266,169.601,36.514,156.873
C06857=1042.105,8.724,-81.251,169.599,36.513,156.873
C06858=1042.098,8.475,-81.236,169.597,36.513,156.872
C06859=1042.093,8.226,-81.221,169.595,36.511,156.872
C06860=1042.086,7.976,-81.206,169.593,36.511,156.872
C06861=1042.079,7.727,-81.190,169.590,36.509,156.872
C06862=1042.073,7.477,-81.175,169.588,36.509,156.872
C06863=1042.067,7.228,-81.160,169.586,36.508,156.871
C06864=1042.061,6.978,-81.144,169.584,36.507,156.871
C06865=1042.054,6.729,-81.129,169.582,36.506,156.871
C06866=1042.048,6.479,-81.114,169.581,36.505,156.871
C06867=1042.042,6.229,-81.099,169.579,36.504,156.871
C06868=1042.035,5.980,-81.084,169.577,36.503,156.871
C06869=1042.029,5.731,-81.069,169.575,36.502,156.871
C06870=1042.022,5.481,-81.054,169.573,36.501,156.870
C06871=1042.016,5.232,-81.039,169.571,36.501,156.870
C06872=1042.010,4.982,-81.024,169.568,36.500,156.870
C06873=1042.003,4.733,-81.009,169.566,36.499,156.870
C06874=1041.997,4.484,-80.994,169.564,36.498,156.870
C06875=1041.991,4.234,-80.978,169.562,36.497,156.869
C06876=1041.985,3.984,-80.963,169.560,36.496,156.869
C06877=1041.979,3.734,-80.948,169.559,36.495,156.869
C06878=1041.972,3.486,-80.933,169.557,36.494,156.869
C06879=1041.966,3.236,-80.918,169.555,36.494,156.869
C06880=1041.960,2.987,-80.903,169.553,36.492,156.869
C06881=1041.953,2.737,-80.888,169.551,36.492,156.869
C06882=1041.947,2.487,-80.873,169.548,36.490,156.868
C06883=1041.941,2.238,-80.858,169.546,36.490,156.868
C06884=1041.934,1.989,-80.843,169.544,36.488,156.868
C06885=1041.928,1.740,-80.828,169.542,36.488,156.868
C06886=1041.922,1.490,-80.813,169.540,36.487,156.868
C06887=1041.915,1.240,-80.798,169.538,36.486,156.868
C06888=1041.909,0.991,-80.783,169.536,36.485,156.867
C06889=1041.903,0.741,-80.768,169.535,36.484,156.867
C06890=1041.897,0.492,-80.753,169.533,36.483,156.867
C06891=1041.891,0.242,-80.738,169.531,36.482,156.867
C06892=1041.885,-0.007,-80.723,169.528,36.481,156.867
C06893=1041.878,-0.257,-80.708,169.526,36.480,156.866
C06894=1041.873,-0.506,-80.694,169.524,36.479,156.866
C06895=1041.866,-0.756,-80.679,169.522,36.479,156.866
C06896=1041.860,-1.005,-80.664,169.520,36.478,156.866
C06897=1041.853,-1.255,-80.649,169.518,36.477,156.866
C06898=1041.848,-1.504,-80.634,169.516,36.476,156.866
C06899=1041.841,-1.754,-80.619,169.514,36.475,156.866
C06900=1041.835,-2.003,-80.604,169.512,36.474,156.865
C06901=1041.828,-2.253,-80.589,169.510,36.473,156.865
C06902=1041.823,-2.502,-80.575,169.508,36.472,156.865
C06903=1041.816,-2.752,-80.560,169.506,36.471,156.865
C06904=1041.809,-3.034,-80.543,169.503,36.470,156.865
C06905=1041.803,-3.318,-80.526,169.501,36.469,156.864
C06906=1041.795,-3.602,-80.508,169.499,36.468,156.864
C06907=1041.788,-3.885,-80.492,169.497,36.467,156.864
C06908=1041.782,-4.134,-80.477,169.495,36.467,156.864
C06909=1041.775,-4.383,-80.463,169.493,36.465,156.864
C06910=1041.769,-4.634,-80.449,169.491,36.465,156.864
C06911=1041.762,-4.883,-80.434,169.489,36.464,156.864
C06912=1041.756,-5.133,-80.419,169.487,36.463,156.863
C06913=1041.749,-5.382,-80.405,169.484,36.462,156.863
C06914=1041.743,-5.631,-80.390,169.482,36.462,156.863
C06915=1041.736,-5.881,-80.375,169.480,36.461,156.863
C06916=1041.730,-6.131,-80.361,169.478,36.460,156.863
C06917=1041.724,-6.380,-80.347,169.476,36.459,156.863
C06918=1041.717,-6.630,-80.332,169.474,36.458,156.863
C06919=1041.711,-6.879,-80.317,169.472,36.458,156.862
C06920=1041.705,-7.128,-80.303,169.470,36.457,156.862
C06921=1041.699,-7.378,-80.289,169.468,36.456,156.862
C06922=1041.692,-7.628,-80.274,169.466,36.455,156.862
C06923=1041.685,-7.877,-80.259,169.464,36.455,156.862
C06924=1041.679,-8.126,-80.245,169.462,36.454,156.862
C06925=1041.673,-8.376,-80.231,169.459,36.453,156.861
C06926=1041.666,-8.626,-80.216,169.457,36.452,156.861
C06927=1041.660,-8.875,-80.202,169.455,36.451,156.861
C06928=1041.654,-9.124,-80.187,169.453,36.451,156.861
C06929=1041.648,-9.375,-80.173,169.451,36.449,156.861
C06930=1041.641,-9.623,-80.159,169.449,36.449,156.861
C06931=1041.635,-9.873,-80.144,169.447,36.448,156.861
C06932=1041.629,-10.123,-80.129,169.445,36.447,156.861
C06933=1041.622,-10.372,-80.115,169.443,36.446,156.860
C06934=1041.616,-10.622,-80.100,169.441,36.446,156.860
C06935=1041.610,-10.872,-80.086,169.439,36.445,156.860
C06936=1041.603,-11.120,-80.072,169.437,36.444,156.860
C06937=1041.597,-11.370,-80.057,169.434,36.443,156.860
C06938=1041.591,-11.620,-80.043,169.432,36.442,156.860
C06939=1041.584,-11.869,-80.029,169.430,36.442,156.860
C06940=1041.578,-12.119,-80.014,169.428,36.441,156.859
C06941=1041.572,-12.368,-80.000,169.426,36.440,156.859
C06942=1041.565,-12.618,-79.986,169.424,36.439,156.859
C06943=1041.560,-12.867,-79.971,169.422,36.438,156.859
C06944=1041.553,-13.117,-79.957,169.420,36.438,156.859
C06945=1041.546,-13.366,-79.943,169.418,36.437,156.859
C06946=1041.541,-13.616,-79.929,169.416,36.436,156.858
C06947=1041.535,-13.865,-79.914,169.414,36.435,156.858
C06948=1041.528,-14.115,-79.901,169.411,36.435,156.858
C06949=1041.522,-14.364,-79.886,169.409,36.433,156.858
C06950=1041.516,-14.613,-79.871,169.407,36.433,156.858
C06951=1041.509,-14.863,-79.858,169.405,36.432,156.858
C06952=1041.503,-15.113,-79.843,169.403,36.431,156.858
C06953=1041.497,-15.362,-79.829,169.401,36.430,156.857
C06954=1041.490,-15.612,-79.814,169.399,36.429,156.857
C06955=1041.484,-15.861,-79.801,169.397,36.429,156.857
C06956=1041.478,-16.111,-79.787,169.395,36.428,156.857
C06957=1041.471,-16.361,-79.773,169.393,36.428,156.857
C06958=1041.465,-16.610,-79.759,169.391,36.427,156.857
C06959=1041.458,-16.860,-79.744,169.389,36.426,156.857
C06960=1041.452,-17.109,-79.731,169.387,36.426,156.857
C06961=1041.446,-17.359,-79.716,169.384,36.425,156.857
C06962=1041.440,-17.608,-79.703,169.382,36.424,156.856
C06963=1041.433,-17.858,-79.689,169.380,36.424,156.856
C06964=1041.427,-18.107,-79.675,169.378,36.422,156.856
C06965=1041.420,-18.357,-79.661,169.375,36.422,156.856
C06966=1041.414,-18.606,-79.646,169.373,36.421,156.856
C06967=1041.407,-18.856,-79.633,169.371,36.420,156.856
C06968=1041.400,-19.137,-79.617,169.369,36.420,156.856
C06969=1041.393,-19.419,-79.602,169.367,36.419,156.856
C06970=1041.387,-19.701,-79.585,169.364,36.418,156.855
C06971=1041.379,-19.984,-79.570,169.362,36.417,156.855
C06972=1041.373,-20.232,-79.556,169.360,36.417,156.855
C06973=1041.366,-20.482,-79.542,169.358,36.416,156.855
C06974=1041.361,-20.732,-79.528,169.355,36.415,156.855
C06975=1041.353,-20.981,-79.514,169.353,36.415,156.855
C06976=1041.348,-21.231,-79.500,169.351,36.414,156.855
C06977=1041.341,-21.481,-79.486,169.349,36.413,156.854
C06978=1041.335,-21.729,-79.472,169.347,36.413,156.854
C06979=1041.329,-21.980,-79.458,169.344,36.411,156.854
C06980=1041.322,-22.229,-79.445,169.342,36.411,156.854
C06981=1041.316,-22.478,-79.431,169.340,36.410,156.854
C06982=1041.310,-22.728,-79.417,169.338,36.409,156.854
C06983=1041.303,-22.977,-79.403,169.336,36.409,156.854
C06984=1041.297,-23.228,-79.389,169.334,36.408,156.854
C06985=1041.291,-23.477,-79.376,169.332,36.408,156.853
C06986=1041.284,-23.726,-79.361,169.330,36.407,156.853
C06987=1041.279,-23.976,-79.348,169.328,36.406,156.853
C06988=1041.272,-24.226,-79.334,169.326,36.406,156.853
C06989=1041.266,-24.475,-79.321,169.323,36.405,156.853
C06990=1041.260,-24.724,-79.307,169.321,36.404,156.853
C06991=1041.253,-24.974,-79.292,169.319,36.403,156.853
C06992=1041.247,-25.223,-79.279,169.317,36.402,156.853
C06993=1041.241,-25.473,-79.265,169.314,36.402,156.852
C06994=1041.234,-25.723,-79.252,169.312,36.401,156.852
C06995=1041.228,-25.972,-79.238,169.310,36.400,156.852
C06996=1041.222,-26.222,-79.224,169.308,36.400,156.852
C06997=1041.216,-26.471,-79.211,169.306,36.399,156.852
C06998=1041.210,-26.720,-79.196,169.304,36.398,156.852
C06999=1041.203,-26.970,-79.183,169.302,36.398,156.852
C07000=1041.197,-27.220,-79.169,169.300,36.397,156.852
C07001=1041.190,-27.470,-79.156,169.298,36.397,156.852
C07002=1041.184,-27.719,-79.142,169.296,36.396,156.851
C07003=1041.178,-27.968,-79.129,169.292,36.395,156.851
C07004=1041.171,-28.218,-79.116,169.290,36.395,156.851
C07005=1041.166,-28.468,-79.102,169.288,36.394,156.851
C07006=1041.159,-28.717,-79.088,169.286,36.393,156.851
C07007=1041.153,-28.967,-79.075,169.284,36.393,156.851
C07008=1041.146,-29.216,-79.062,169.282,36.392,156.851
C07009=1041.140,-29.466,-79.048,169.280,36.392,156.851
C07010=1041.133,-29.715,-79.035,169.278,36.391,156.851
C07011=1041.127,-29.965,-79.021,169.275,36.391,156.851
C07012=1041.120,-30.215,-79.008,169.273,36.390,156.850
C07013=1041.114,-30.464,-78.994,169.271,36.389,156.850
C07014=1041.109,-30.713,-78.981,169.269,36.389,156.850
C07015=1041.102,-30.963,-78.967,169.267,36.388,156.850
C07016=1041.096,-31.213,-78.954,169.265,36.387,156.850
C07017=1041.089,-31.462,-78.940,169.263,36.387,156.850
C07018=1041.083,-31.712,-78.927,169.260,36.386,156.850
C07019=1041.077,-31.962,-78.914,169.257,36.386,156.850
C07020=1041.070,-32.211,-78.901,169.255,36.385,156.849
C07021=1041.064,-32.461,-78.887,169.253,36.385,156.849
C07022=1041.057,-32.710,-78.874,169.251,36.384,156.849
C07023=1041.051,-32.960,-78.861,169.249,36.384,156.849
C07024=1041.045,-33.209,-78.848,169.247,36.383,156.849
C07025=1041.038,-33.459,-78.834,169.244,36.382,156.849
C07026=1041.032,-33.708,-78.821,169.242,36.382,156.849
C07027=1041.027,-33.958,-78.807,169.240,36.381,156.849
C07028=1041.021,-34.207,-78.794,169.238,36.380,156.849
C07029=1041.014,-34.457,-78.781,169.236,36.380,156.849
C07030=1041.008,-34.707,-78.767,169.234,36.379,156.848
C07031=1041.001,-34.956,-78.754,169.232,36.379,156.848
C07032=1040.994,-35.237,-78.740,169.229,36.378,156.848
C07033=1040.987,-35.519,-78.724,169.227,36.378,156.848
C07034=1040.980,-35.799,-78.710,169.224,36.377,156.848
C07035=1040.973,-36.080,-78.695,169.221,36.376,156.848
C07036=1040.967,-36.330,-78.682,169.219,36.376,156.848
C07037=1040.961,-36.579,-78.669,169.217,36.375,156.848
C07038=1040.954,-36.829,-78.655,169.214,36.374,156.848
C07039=1040.948,-37.079,-78.641,169.212,36.374,156.848
C07040=1040.942,-37.329,-78.629,169.210,36.373,156.847
C07041=1040.936,-37.578,-78.615,169.208,36.372,156.847
C07042=1040.930,-37.827,-78.602,169.206,36.372,156.847
C07043=1040.923,-38.077,-78.589,169.204,36.371,156.847
C07044=1040.917,-38.327,-78.576,169.201,36.371,156.847
C07045=1040.911,-38.576,-78.563,169.199,36.371,156.847
C07046=1040.905,-38.825,-78.549,169.197,36.370,156.847
C07047=1040.899,-39.075,-78.537,169.195,36.369,156.847
C07048=1040.891,-39.325,-78.524,169.193,36.369,156.847
C07049=1040.885,-39.575,-78.511,169.190,36.369,156.847
C07050=1040.879,-39.824,-78.498,169.188,36.368,156.847
C07051=1040.873,-40.073,-78.485,169.186,36.367,156.846
C07052=1040.867,-40.323,-78.472,169.184,36.367,156.846
C07053=1040.859,-40.573,-78.459,169.182,36.367,156.846
C07054=1040.854,-40.823,-78.447,169.179,36.366,156.846
C07055=1040.847,-41.072,-78.433,169.176,36.365,156.846
C07056=1040.841,-41.321,-78.420,169.174,36.365,156.846
C07057=1040.835,-41.571,-78.408,169.172,36.365,156.846
C07058=1040.828,-41.820,-78.395,169.170,36.364,156.846
C07059=1040.822,-42.071,-78.382,169.167,36.363,156.846
C07060=1040.816,-42.320,-78.369,169.165,36.363,156.846
C07061=1040.810,-42.570,-78.356,169.163,36.363,156.846
C07062=1040.803,-42.819,-78.343,169.161,36.362,156.846
C07063=1040.797,-43.069,-78.331,169.159,36.361,156.845
C07064=1040.791,-43.318,-78.318,169.156,36.361,156.845
C07065=1040.785,-43.568,-78.305,169.154,36.361,156.845
C07066=1040.778,-43.817,-78.292,169.152,36.360,156.845
C07067=1040.771,-44.067,-78.279,169.150,36.360,156.845
C07068=1040.765,-44.317,-78.266,169.147,36.359,156.845
C07069=1040.759,-44.567,-78.254,169.145,36.359,156.845
C07070=1040.753,-44.816,-78.240,169.143,36.358,156.845
C07071=1040.747,-45.066,-78.228,169.141,36.358,156.845
C07072=1040.740,-45.315,-78.215,169.139,36.357,156.845
C07073=1040.734,-45.565,-78.203,169.136,36.357,156.845
C07074=1040.728,-45.815,-78.190,169.134,36.357,156.845
C07075=1040.722,-46.064,-78.177,169.132,36.356,156.845
C07076=1040.715,-46.313,-78.165,169.130,36.355,156.844
C07077=1040.709,-46.563,-78.152,169.127,36.355,156.844
C07078=1040.703,-46.812,-78.139,169.124,36.355,156.844
C07079=1040.697,-47.062,-78.126,169.122,36.354,156.844
C07080=1040.690,-47.311,-78.114,169.120,36.353,156.844
C07081=1040.684,-47.561,-78.101,169.117,36.353,156.844
C07082=1040.679,-47.811,-78.089,169.115,36.353,156.844
C07083=1040.672,-48.060,-78.075,169.113,36.352,156.844
C07084=1040.666,-48.310,-78.063,169.111,36.352,156.844
C07085=1040.660,-48.560,-78.051,169.109,36.352,156.844
C07086=1040.654,-48.809,-78.038,169.106,36.351,156.844
C07087=1040.648,-49.059,-78.025,169.104,36.351,156.844
C07088=1040.641,-49.309,-78.013,169.102,36.350,156.844
C07089=1040.635,-49.558,-78.000,169.100,36.350,156.843
C07090=1040.629,-49.808,-77.987,169.097,36.350,156.843
C07091=1040.622,-50.057,-77.975,169.095,36.349,156.843
C07092=1040.616,-50.307,-77.963,169.093,36.348,156.843
C07093=1040.610,-50.556,-77.950,169.091,36.348,156.843
C07094=1040.603,-50.806,-77.938,169.088,36.348,156.843
C07095=1040.597,-51.057,-77.925,169.086,36.348,156.843
C07096=1040.589,-51.337,-77.911,169.083,36.347,156.843
C07097=1040.582,-51.619,-77.897,169.081,36.347,156.843
C07098=1040.575,-51.900,-77.883,169.078,36.346,156.843
C07099=1040.568,-52.182,-77.869,169.076,36.346,156.843
C07100=1040.561,-52.432,-77.857,169.073,36.346,156.843
C07101=1040.555,-52.682,-77.845,169.071,36.346,156.843
C07102=1040.548,-52.931,-77.832,169.069,36.345,156.843
C07103=1040.542,-53.180,-77.820,169.066,36.345,156.843
C07104=1040.536,-53.430,-77.808,169.064,36.345,156.843
C07105=1040.529,-53.680,-77.796,169.061,36.344,156.843
C07106=1040.523,-53.929,-77.784,169.059,36.344,156.843
C07107=1040.517,-54.179,-77.771,169.056,36.344,156.842
C07108=1040.511,-54.428,-77.760,169.054,36.344,156.842
C07109=1040.505,-54.678,-77.747,169.052,36.343,156.842
C07110=1040.498,-54.928,-77.735,169.049,36.343,156.842
C07111=1040.491,-55.177,-77.723,169.047,36.343,156.842
C07112=1040.486,-55.427,-77.711,169.045,36.342,156.842
C07113=1040.479,-55.677,-77.699,169.042,36.342,156.842
C07114=1040.472,-55.926,-77.687,169.040,36.342,156.842
C07115=1040.466,-56.176,-77.674,169.038,36.342,156.842
C07116=1040.460,-56.426,-77.662,169.035,36.342,156.842
C07117=1040.453,-56.675,-77.650,169.033,36.341,156.842
C07118=1040.447,-56.925,-77.638,169.031,36.341,156.842
C07119=1040.441,-57.175,-77.626,169.028,36.340,156.842
C07120=1040.435,-57.425,-77.613,169.026,36.340,156.842
C07121=1040.429,-57.674,-77.601,169.024,36.340,156.842
C07122=1040.422,-57.923,-77.589,169.021,36.340,156.842
C07123=1040.416,-58.173,-77.577,169.019,36.340,156.842
C07124=1040.409,-58.423,-77.565,169.017,36.339,156.842
C07125=1040.403,-58.672,-77.553,169.015,36.339,156.842
C07126=1040.397,-58.922,-77.540,169.012,36.339,156.842
C07127=1040.390,-59.172,-77.529,169.010,36.338,156.842
C07128=1040.384,-59.421,-77.517,169.008,36.338,156.842
C07129=1040.378,-59.670,-77.504,169.005,36.338,156.841
C07130=1040.372,-59.921,-77.493,169.003,36.338,156.841
C07131=1040.365,-60.170,-77.481,169.001,36.338,156.841
C07132=1040.359,-60.420,-77.469,168.998,36.337,156.841
C07133=1040.353,-60.670,-77.457,168.996,36.337,156.841
C07134=1040.346,-60.919,-77.445,168.994,36.337,156.841
C07135=1040.340,-61.168,-77.433,168.991,36.336,156.841
C07136=1040.334,-61.418,-77.421,168.989,36.336,156.841
C07137=1040.328,-61.668,-77.409,168.987,36.335,156.841
C07138=1040.321,-61.918,-77.397,168.984,36.335,156.841
C07139=1040.316,-62.167,-77.385,168.982,36.335,156.841
C07140=1040.309,-62.416,-77.373,168.980,36.335,156.841
C07141=1040.302,-62.666,-77.361,168.977,36.335,156.841
C07142=1040.297,-62.916,-77.349,168.975,36.335,156.841
C07143=1040.290,-63.166,-77.337,168.973,36.334,156.841
C07144=1040.284,-63.415,-77.326,168.970,36.334,156.841
C07145=1040.278,-63.665,-77.313,168.968,36.334,156.841
C07146=1040.272,-63.914,-77.301,168.965,36.333,156.841
C07147=1040.265,-64.165,-77.290,168.962,36.333,156.841
C07148=1040.259,-64.413,-77.278,168.960,36.333,156.841
C07149=1040.253,-64.663,-77.266,168.957,36.333,156.841
C07150=1040.247,-64.913,-77.254,168.955,36.333,156.841
C07151=1040.240,-65.163,-77.243,168.953,36.333,156.841
C07152=1040.234,-65.412,-77.231,168.950,36.332,156.841
C07153=1040.228,-65.662,-77.219,168.948,36.332,156.841
C07154=1040.222,-65.912,-77.207,168.946,36.332,156.841
C07155=1040.216,-66.161,-77.196,168.943,36.331,156.841
C07156=1040.210,-66.411,-77.183,168.941,36.331,156.841
C07157=1040.204,-66.661,-77.172,168.939,36.331,156.841
C07158=1040.198,-66.910,-77.160,168.936,36.331,156.840
C07159=1040.191,-67.159,-77.148,168.934,36.331,156.840
C07160=1040.183,-67.478,-77.133,168.931,36.331,156.840
C07161=1040.176,-67.796,-77.118,168.928,36.330,156.840
C07162=1040.168,-68.114,-77.104,168.925,36.330,156.840
C07163=1040.160,-68.433,-77.089,168.922,36.329,156.840
C07164=1040.154,-68.682,-77.077,168.920,36.329,156.840
C07165=1040.148,-68.932,-77.066,168.917,36.329,156.840
C07166=1040.141,-69.182,-77.054,168.915,36.329,156.840
C07167=1040.136,-69.431,-77.042,168.913,36.329,156.840
C07168=1040.130,-69.681,-77.030,168.910,36.329,156.840
C07169=1040.124,-69.930,-77.019,168.908,36.328,156.840
C07170=1040.117,-70.180,-77.008,168.905,36.328,156.840
C07171=1040.111,-70.430,-76.995,168.903,36.328,156.840
C07172=1040.106,-70.680,-76.984,168.901,36.328,156.840
C07173=1040.099,-70.929,-76.972,168.898,36.327,156.840
C07174=1040.093,-71.179,-76.961,168.896,36.327,156.840
C07175=1040.087,-71.429,-76.949,168.894,36.327,156.840
C07176=1040.081,-71.679,-76.937,168.891,36.327,156.840
C07177=1040.075,-71.928,-76.926,168.889,36.327,156.840
C07178=1040.069,-72.178,-76.915,168.886,36.327,156.840
C07179=1040.062,-72.427,-76.903,168.884,36.327,156.840
C07180=1040.057,-72.677,-76.891,168.882,36.326,156.840
C07181=1040.051,-72.926,-76.880,168.879,36.326,156.840
C07182=1040.044,-73.176,-76.868,168.877,36.326,156.840
C07183=1040.038,-73.425,-76.857,168.875,36.326,156.840
C07184=1040.033,-73.658,-76.846,168.872,36.325,156.840
C07185=1040.027,-73.890,-76.836,168.870,36.325,156.840
C07186=1040.022,-74.122,-76.824,168.868,36.325,156.840
C07187=1040.016,-74.354,-76.814,168.866,36.325,156.840
C07188=1040.010,-74.585,-76.804,168.863,36.325,156.840
C07189=1040.004,-74.818,-76.793,168.861,36.325,156.840
C07190=1039.998,-75.049,-76.783,168.859,36.325,156.840
C07191=1039.993,-75.282,-76.772,168.857,36.325,156.840
C07192=1039.987,-75.531,-76.761,168.854,36.325,156.839
C07193=1039.980,-75.781,-76.749,168.852,36.325,156.839
C07194=1039.974,-76.030,-76.739,168.849,36.324,156.839
C07195=1039.968,-76.280,-76.727,168.847,36.324,156.839
C07196=1039.962,-76.530,-76.716,168.845,36.324,156.839
C07197=1039.955,-76.779,-76.704,168.842,36.324,156.840
C07198=1039.949,-77.029,-76.694,168.840,36.324,156.840
C07199=1039.943,-77.279,-76.682,168.837,36.324,156.840
C07200=1039.937,-77.528,-76.671,168.835,36.324,156.840
C07201=1039.931,-77.778,-76.660,168.832,36.324,156.840
C07202=1039.925,-78.027,-76.649,168.830,36.324,156.840
C07203=1039.919,-78.278,-76.637,168.828,36.324,156.840
C07204=1039.913,-78.527,-76.627,168.825,36.324,156.840
C07205=1039.906,-78.777,-76.615,168.823,36.324,156.840
C07206=1039.900,-79.026,-76.604,168.820,36.324,156.840
C07207=1039.894,-79.276,-76.592,168.818,36.324,156.840
C07208=1039.888,-79.526,-76.582,168.815,36.324,156.840
C07209=1039.882,-79.776,-76.570,168.813,36.324,156.840
C07210=1039.876,-80.025,-76.560,168.811,36.324,156.840
C07211=1039.869,-80.275,-76.548,168.808,36.324,156.840
C07212=1039.863,-80.524,-76.537,168.806,36.324,156.840
C07213=1039.856,-80.774,-76.527,168.803,36.324,156.840
C07214=1039.850,-81.024,-76.516,168.801,36.324,156.840
C07215=1039.844,-81.274,-76.504,168.798,36.324,156.840
C07216=1039.838,-81.523,-76.494,168.796,36.324,156.840
C07217=1039.832,-81.772,-76.483,168.793,36.325,156.840
C07218=1039.825,-82.023,-76.472,168.791,36.325,156.840
C07219=1039.820,-82.272,-76.461,168.788,36.325,156.840
C07220=1039.813,-82.522,-76.450,168.786,36.325,156.840
C07221=1039.807,-82.771,-76.440,168.783,36.325,156.840
C07222=1039.801,-83.022,-76.428,168.781,36.325,156.840
C07223=1039.794,-83.271,-76.418,168.778,36.325,156.840
C07224=1039.786,-83.556,-76.405,168.776,36.325,156.840
C07225=1039.780,-83.840,-76.393,168.773,36.325,156.840
C07226=1039.772,-84.126,-76.381,168.770,36.325,156.840
